# B&R Automation Studio project TD52 (part 112)

#### MsgGTInit.st - Cyclic code
```iecst
(*******************************************************************************
Msg_VE	 			 alarms generation MM_ventilation

This code is confidential and proprietary to the INNIO Company.
It may not be used in any form, or reproduced in any manner,
without written permission of the INNIO Company.
Copyright, INNIO Company, 2019

Customized modifications: -
------------------------

History:
-------
V0.00.0	29.07.2011	lettenb.	new

Instructions for use:
--------------------
1) declare alarm with function block "Msg"

2) use template to create a new alarm, substitue 0000 by message number:

	xMsg0000.Num		:=	0000;					alarm number
	xMsg0000.AmmSysAdr	:=  iAdrAmmBase2MM;			do not change
	xMsg0000.AmmOutAdr	:=  iAdrMM2AmmBase;			do not change

3) 	set alarm number

Outstandings:
------------
(*******************************************************************************)
PROGRAM _INIT

	iAdrAmmBase2MM		:=  ADR(IN_GT.tAB2GT);
	iAdrMM2AmmBase		:=  ADR(OUT_GT.tGT2AB);

	(*---------------------------------------------------------------------------*)
	xMsg1027.Num		:=  1027;
	xMsg1027.AmmInAdr	:=  iAdrAmmBase2MM;
	xMsg1027.AmmOutAdr	:=  iAdrMM2AmmBase;

	xMsg1028.Num		:=  1028;
	xMsg1028.AmmInAdr	:=  iAdrAmmBase2MM;
	xMsg1028.AmmOutAdr	:=  iAdrMM2AmmBase;

	xMsg1029.Num		:=  1029;
	xMsg1029.AmmInAdr	:=  iAdrAmmBase2MM;
	xMsg1029.AmmOutAdr	:=  iAdrMM2AmmBase;

	xMsg1030.Num		:=  1030;
	xMsg1030.AmmInAdr	:=  iAdrAmmBase2MM;
	xMsg1030.AmmOutAdr	:=  iAdrMM2AmmBase;

	xMsg1057.Num		:=  1057;
	xMsg1057.AmmInAdr	:=  iAdrAmmBase2MM;
	xMsg1057.AmmOutAdr	:=  iAdrMM2AmmBase;

	xMsg1058.Num		:=  1058;
	xMsg1058.AmmInAdr	:=  iAdrAmmBase2MM;
	xMsg1058.AmmOutAdr	:=  iAdrMM2AmmBase;

	xMsg1084.Num		:=  1084;
	xMsg1084.AmmInAdr	:=  iAdrAmmBase2MM;
	xMsg1084.AmmOutAdr	:=  iAdrMM2AmmBase;

	xMsg1085.Num		:=  1085;
	xMsg1085.AmmInAdr	:=  iAdrAmmBase2MM;
	xMsg1085.AmmOutAdr	:=  iAdrMM2AmmBase;

	xMsg1086.Num		:=  1086;
	xMsg1086.AmmInAdr	:=  iAdrAmmBase2MM;
	xMsg1086.AmmOutAdr	:=  iAdrMM2AmmBase;

	xMsg1087.Num		:=  1087;
	xMsg1087.AmmInAdr	:=  iAdrAmmBase2MM;
	xMsg1087.AmmOutAdr	:=  iAdrMM2AmmBase;

	xMsg1088.Num		:=  1088;
	xMsg1088.AmmInAdr	:=  iAdrAmmBase2MM;
	xMsg1088.AmmOutAdr	:=  iAdrMM2AmmBase;

	xMsg1094.Num		:=  1094;
	xMsg1094.AmmInAdr	:=  iAdrAmmBase2MM;
	xMsg1094.AmmOutAdr	:=  iAdrMM2AmmBase;

	xMsg1095.Num		:=  1095;
	xMsg1095.AmmInAdr	:=  iAdrAmmBase2MM;
	xMsg1095.AmmOutAdr	:=  iAdrMM2AmmBase;

	xMsg1128.Num		:=  1128;
	xMsg1128.AmmInAdr	:=  iAdrAmmBase2MM;
	xMsg1128.AmmOutAdr	:=  iAdrMM2AmmBase;

	xMsg1251.Num		:=  1251;
	xMsg1251.AmmInAdr	:=  iAdrAmmBase2MM;
	xMsg1251.AmmOutAdr	:=  iAdrMM2AmmBase;

	xMsg1252.Num		:=  1252;
	xMsg1252.AmmInAdr	:=  iAdrAmmBase2MM;
	xMsg1252.AmmOutAdr	:=  iAdrMM2AmmBase;

	xMsg2243.Num		:=  2243;
	xMsg2243.AmmInAdr	:=  iAdrAmmBase2MM;
	xMsg2243.AmmOutAdr	:=  iAdrMM2AmmBase;

	xMsg2246.Num		:=  2246;
	xMsg2246.AmmInAdr	:=  iAdrAmmBase2MM;
	xMsg2246.AmmOutAdr	:=  iAdrMM2AmmBase;

	xMsg2247.Num		:=  2247;
	xMsg2247.AmmInAdr	:=  iAdrAmmBase2MM;
	xMsg2247.AmmOutAdr	:=  iAdrMM2AmmBase;

	xMsg2250.Num		:=  2250;
	xMsg2250.AmmInAdr	:=  iAdrAmmBase2MM;
	xMsg2250.AmmOutAdr	:=  iAdrMM2AmmBase;

	xMsg2251.Num		:=  2251;
	xMsg2251.AmmInAdr	:=  iAdrAmmBase2MM;
	xMsg2251.AmmOutAdr	:=  iAdrMM2AmmBase;

	xMsg2257.Num		:=  2257;
	xMsg2257.AmmInAdr	:=  iAdrAmmBase2MM;
	xMsg2257.AmmOutAdr	:=  iAdrMM2AmmBase;

	xMsg2535.Num		:=  2535;
	xMsg2535.AmmInAdr	:=  iAdrAmmBase2MM;
	xMsg2535.AmmOutAdr	:=  iAdrMM2AmmBase;

	xMsg2536.Num		:=  2536;
	xMsg2536.AmmInAdr	:=  iAdrAmmBase2MM;
	xMsg2536.AmmOutAdr	:=  iAdrMM2AmmBase;

	xMsg2537.Num		:=  2537;
	xMsg2537.AmmInAdr	:=  iAdrAmmBase2MM;
	xMsg2537.AmmOutAdr	:=  iAdrMM2AmmBase;

	xMsg2538.Num		:=  2538;
	xMsg2538.AmmInAdr	:=  iAdrAmmBase2MM;
	xMsg2538.AmmOutAdr	:=  iAdrMM2AmmBase;

	xMsg2578.Num		:=  2578;
	xMsg2578.AmmInAdr	:=  iAdrAmmBase2MM;
	xMsg2578.AmmOutAdr	:=  iAdrMM2AmmBase;

	xMsg2674.Num		:=  2674;
	xMsg2674.AmmInAdr	:=  iAdrAmmBase2MM;
	xMsg2674.AmmOutAdr	:=  iAdrMM2AmmBase;

	xMsg3004.Num		:=  3004;
	xMsg3004.AmmInAdr	:=  iAdrAmmBase2MM;
	xMsg3004.AmmOutAdr	:=  iAdrMM2AmmBase;

	xMsg3153.Num		:=  3153;
	xMsg3153.AmmInAdr	:=  iAdrAmmBase2MM;
	xMsg3153.AmmOutAdr	:=  iAdrMM2AmmBase;

	xMsg3154.Num		:=  3154;
	xMsg3154.AmmInAdr	:=  iAdrAmmBase2MM;
	xMsg3154.AmmOutAdr	:=  iAdrMM2AmmBase;

	xMsg3155.Num		:=  3155;
	xMsg3155.AmmInAdr	:=  iAdrAmmBase2MM;
	xMsg3155.AmmOutAdr	:=  iAdrMM2AmmBase;

	xMsg3156.Num		:=  3156;
	xMsg3156.AmmInAdr	:=  iAdrAmmBase2MM;
	xMsg3156.AmmOutAdr	:=  iAdrMM2AmmBase;

	xMsg3157.Num		:=  3157;
	xMsg3157.AmmInAdr	:=  iAdrAmmBase2MM;
	xMsg3157.AmmOutAdr	:=  iAdrMM2AmmBase;

	xMsg3158.Num		:=  3158;
	xMsg3158.AmmInAdr	:=  iAdrAmmBase2MM;
	xMsg3158.AmmOutAdr	:=  iAdrMM2AmmBase;

	xMsg3159.Num		:=  3159;
	xMsg3159.AmmInAdr	:=  iAdrAmmBase2MM;
	xMsg3159.AmmOutAdr	:=  iAdrMM2AmmBase;

	xMsg3160.Num		:=  3160;
	xMsg3160.AmmInAdr	:=  iAdrAmmBase2MM;
	xMsg3160.AmmOutAdr	:=  iAdrMM2AmmBase;

	xMsg3221.Num		:=  3221;
	xMsg3221.AmmInAdr	:=  iAdrAmmBase2MM;
	xMsg3221.AmmOutAdr	:=  iAdrMM2AmmBase;

	xMsg3222.Num		:=  3222;
	xMsg3222.AmmInAdr	:=  iAdrAmmBase2MM;
	xMsg3222.AmmOutAdr	:=  iAdrMM2AmmBase;

	xMsg3227.Num		:=	3227;
	xMsg3227.AmmInAdr	:=  iAdrAmmBase2MM;
	xMsg3227.AmmOutAdr	:=  iAdrMM2AmmBase;

	xMsg3257.Num		:=	3257;
	xMsg3257.AmmInAdr	:=  iAdrAmmBase2MM;
	xMsg3257.AmmOutAdr	:=  iAdrMM2AmmBase;

	xMsg3258.Num		:=	3258;
	xMsg3258.AmmInAdr	:=  iAdrAmmBase2MM;
	xMsg3258.AmmOutAdr	:=  iAdrMM2AmmBase;

	xMsg3259.Num		:=	3259;
	xMsg3259.AmmInAdr	:=  iAdrAmmBase2MM;
	xMsg3259.AmmOutAdr	:=  iAdrMM2AmmBase;

	xMsg3260.Num		:=	3260;
	xMsg3260.AmmInAdr	:=  iAdrAmmBase2MM;
	xMsg3260.AmmOutAdr	:=  iAdrMM2AmmBase;

	xMsg3261.Num		:=	3261;
	xMsg3261.AmmInAdr	:=  iAdrAmmBase2MM;
	xMsg3261.AmmOutAdr	:=  iAdrMM2AmmBase;

	xMsg3262.Num		:=	3262;
	xMsg3262.AmmInAdr	:=  iAdrAmmBase2MM;
	xMsg3262.AmmOutAdr	:=  iAdrMM2AmmBase;

	xMsg3308.Num		:=  3308;
	xMsg3308.AmmInAdr	:=  iAdrAmmBase2MM;
	xMsg3308.AmmOutAdr	:=  iAdrMM2AmmBase;

	xMsg3309.Num		:=  3309;
	xMsg3309.AmmInAdr	:=  iAdrAmmBase2MM;
	xMsg3309.AmmOutAdr	:=  iAdrMM2AmmBase;

	xMsg3315.Num		:=  3315;
	xMsg3315.AmmInAdr	:=  iAdrAmmBase2MM;
	xMsg3315.AmmOutAdr	:=  iAdrMM2AmmBase;

	xMsg3316.Num		:=  3316;
	xMsg3316.AmmInAdr	:=  iAdrAmmBase2MM;
	xMsg3316.AmmOutAdr	:=  iAdrMM2AmmBase;

	xMsg3317.Num		:=  3317;
	xMsg3317.AmmInAdr	:=  iAdrAmmBase2MM;
	xMsg3317.AmmOutAdr	:=  iAdrMM2AmmBase;

	xMsg3318.Num		:=  3318;
	xMsg3318.AmmInAdr	:=  iAdrAmmBase2MM;
	xMsg3318.AmmOutAdr	:=  iAdrMM2AmmBase;

	xMsg3320.Num		:=  3320;
	xMsg3320.AmmInAdr	:=  iAdrAmmBase2MM;
	xMsg3320.AmmOutAdr	:=  iAdrMM2AmmBase;

	xMsg3324.Num		:=  3324;
	xMsg3324.AmmInAdr	:=  iAdrAmmBase2MM;
	xMsg3324.AmmOutAdr	:=  iAdrMM2AmmBase;

	xMsg3325.Num		:=  3325;
	xMsg3325.AmmInAdr	:=  iAdrAmmBase2MM;
	xMsg3325.AmmOutAdr	:=  iAdrMM2AmmBase;

	xMsg3326.Num		:=  3326;
	xMsg3326.AmmInAdr	:=  iAdrAmmBase2MM;
	xMsg3326.AmmOutAdr	:=  iAdrMM2AmmBase;

	xMsg3327.Num		:=  3327;
	xMsg3327.AmmInAdr	:=  iAdrAmmBase2MM;
	xMsg3327.AmmOutAdr	:=  iAdrMM2AmmBase;

	xMsg3328.Num		:=  3328;
	xMsg3328.AmmInAdr	:=  iAdrAmmBase2MM;
	xMsg3328.AmmOutAdr	:=  iAdrMM2AmmBase;

	xMsg3353.Num		:=  3353;
	xMsg3353.AmmInAdr	:=  iAdrAmmBase2MM;
	xMsg3353.AmmOutAdr	:=  iAdrMM2AmmBase;

	xMsg3354.Num		:=  3354;
	xMsg3354.AmmInAdr	:=  iAdrAmmBase2MM;
	xMsg3354.AmmOutAdr	:=  iAdrMM2AmmBase;

	xMsg3355.Num		:=  3355;
	xMsg3355.AmmInAdr	:=  iAdrAmmBase2MM;
	xMsg3355.AmmOutAdr	:=  iAdrMM2AmmBase;

	xMsg3356.Num		:=  3356;
	xMsg3356.AmmInAdr	:=  iAdrAmmBase2MM;
	xMsg3356.AmmOutAdr	:=  iAdrMM2AmmBase;

	xMsg3357.Num		:=  3357;
	xMsg3357.AmmInAdr	:=  iAdrAmmBase2MM;
	xMsg3357.AmmOutAdr	:=  iAdrMM2AmmBase;

	xMsg3358.Num		:=  3358;
	xMsg3358.AmmInAdr	:=  iAdrAmmBase2MM;
	xMsg3358.AmmOutAdr	:=  iAdrMM2AmmBase;

	xMsg3359.Num		:=  3359;
	xMsg3359.AmmInAdr	:=  iAdrAmmBase2MM;
	xMsg3359.AmmOutAdr	:=  iAdrMM2AmmBase;

	xMsg3360.Num		:=  3360;
	xMsg3360.AmmInAdr	:=  iAdrAmmBase2MM;
	xMsg3360.AmmOutAdr	:=  iAdrMM2AmmBase;

	xMsg3361.Num		:=  3361;
	xMsg3361.AmmInAdr	:=  iAdrAmmBase2MM;
	xMsg3361.AmmOutAdr	:=  iAdrMM2AmmBase;

	xMsg3362.Num		:=  3362;
	xMsg3362.AmmInAdr	:=  iAdrAmmBase2MM;
	xMsg3362.AmmOutAdr	:=  iAdrMM2AmmBase;

	xMsg3363.Num		:=  3363;
	xMsg3363.AmmInAdr	:=  iAdrAmmBase2MM;
	xMsg3363.AmmOutAdr	:=  iAdrMM2AmmBase;

	xMsg3364.Num		:=  3364;
	xMsg3364.AmmInAdr	:=  iAdrAmmBase2MM;
	xMsg3364.AmmOutAdr	:=  iAdrMM2AmmBase;

	xMsg3365.Num		:=  3365;
	xMsg3365.AmmInAdr	:=  iAdrAmmBase2MM;
	xMsg3365.AmmOutAdr	:=  iAdrMM2AmmBase;

	xMsg3520.Num		:=  3520;
	xMsg3520.AmmInAdr	:=  iAdrAmmBase2MM;
	xMsg3520.AmmOutAdr	:=  iAdrMM2AmmBase;

	xMsg3567.Num		:=  3567;
	xMsg3567.AmmInAdr	:=  iAdrAmmBase2MM;
	xMsg3567.AmmOutAdr	:=  iAdrMM2AmmBase;

	xMsg3568.Num		:=  3568;
	xMsg3568.AmmInAdr	:=  iAdrAmmBase2MM;
	xMsg3568.AmmOutAdr	:=  iAdrMM2AmmBase;

	xMsg3569.Num		:=  3569;
	xMsg3569.AmmInAdr	:=  iAdrAmmBase2MM;
	xMsg3569.AmmOutAdr	:=  iAdrMM2AmmBase;

	xMsg3570.Num		:=  3570;
	xMsg3570.AmmInAdr	:=  iAdrAmmBase2MM;
	xMsg3570.AmmOutAdr	:=  iAdrMM2AmmBase;

	xMsg3525.Num		:=  3525;
	xMsg3525.AmmInAdr	:=  iAdrAmmBase2MM;
	xMsg3525.AmmOutAdr	:=  iAdrMM2AmmBase;

	xMsg2247.Num		:=  2247;
	xMsg2247.AmmInAdr	:=  iAdrAmmBase2MM;
	xMsg2247.AmmOutAdr	:=  iAdrMM2AmmBase;

	xMsg2257.Num		:=  2257;
	xMsg2257.AmmInAdr	:=  iAdrAmmBase2MM;
	xMsg2257.AmmOutAdr	:=  iAdrMM2AmmBase;

	xMsg3448.Num		:=  3448;
	xMsg3448.AmmInAdr	:=  iAdrAmmBase2MM;
	xMsg3448.AmmOutAdr	:=  iAdrMM2AmmBase;

	xMsg3444.Num		:=  3444;
	xMsg3444.AmmInAdr	:=  iAdrAmmBase2MM;
	xMsg3444.AmmOutAdr	:=  iAdrMM2AmmBase;

	xMsg3376.Num		:=  3376;
	xMsg3376.AmmInAdr	:=  iAdrAmmBase2MM;
	xMsg3376.AmmOutAdr	:=  iAdrMM2AmmBase;

	xMsg3445.Num		:=  3445;
	xMsg3445.AmmInAdr	:=  iAdrAmmBase2MM;
	xMsg3445.AmmOutAdr	:=  iAdrMM2AmmBase;

	xMsg2289.Num		:=  2289;
	xMsg2289.AmmInAdr	:=  iAdrAmmBase2MM;
	xMsg2289.AmmOutAdr	:=  iAdrMM2AmmBase;

	xMsg2271.Num		:=  2271;
	xMsg2271.AmmInAdr	:=  iAdrAmmBase2MM;
	xMsg2271.AmmOutAdr	:=  iAdrMM2AmmBase;

	xMsg2261.Num		:=  2261;
	xMsg2261.AmmInAdr	:=  iAdrAmmBase2MM;
	xMsg2261.AmmOutAdr	:=  iAdrMM2AmmBase;

	xMsg3377.Num		:=  3377;
	xMsg3377.AmmInAdr	:=  iAdrAmmBase2MM;
	xMsg3377.AmmOutAdr	:=  iAdrMM2AmmBase;

	xMsg2272.Num		:=  2272;
	xMsg2272.AmmInAdr	:=  iAdrAmmBase2MM;
	xMsg2272.AmmOutAdr	:=  iAdrMM2AmmBase;

	xMsg2231.Num		:=  2231;
	xMsg2231.AmmInAdr	:=  iAdrAmmBase2MM;
	xMsg2231.AmmOutAdr	:=  iAdrMM2AmmBase;

	xMsg2240.Num		:=  2240;
	xMsg2240.AmmInAdr	:=  iAdrAmmBase2MM;
	xMsg2240.AmmOutAdr	:=  iAdrMM2AmmBase;

	xMsg2241.Num		:=  2241;
	xMsg2241.AmmInAdr	:=  iAdrAmmBase2MM;
	xMsg2241.AmmOutAdr	:=  iAdrMM2AmmBase;

	xMsg2248.Num		:=  2248;
	xMsg2248.AmmInAdr	:=  iAdrAmmBase2MM;
	xMsg2248.AmmOutAdr	:=  iAdrMM2AmmBase;

	xMsg2249.Num		:=  2249;
	xMsg2249.AmmInAdr	:=  iAdrAmmBase2MM;
	xMsg2249.AmmOutAdr	:=  iAdrMM2AmmBase;

	xMsg2273.Num		:=  2273;
	xMsg2273.AmmInAdr	:=  iAdrAmmBase2MM;
	xMsg2273.AmmOutAdr	:=  iAdrMM2AmmBase;

	xMsg2567.Num		:=  2567;
	xMsg2567.AmmInAdr	:=  iAdrAmmBase2MM;
	xMsg2567.AmmOutAdr	:=  iAdrMM2AmmBase;

	xMsg2568.Num		:=  2568;
	xMsg2568.AmmInAdr	:=  iAdrAmmBase2MM;
	xMsg2568.AmmOutAdr	:=  iAdrMM2AmmBase;

	xMsg2569.Num		:=  2569;
	xMsg2569.AmmInAdr	:=  iAdrAmmBase2MM;
	xMsg2569.AmmOutAdr	:=  iAdrMM2AmmBase;

	xMsg2580.Num		:=  2580;
	xMsg2580.AmmInAdr	:=  iAdrAmmBase2MM;
	xMsg2580.AmmOutAdr	:=  iAdrMM2AmmBase;

	xMsg2581.Num		:=  2581;
	xMsg2581.AmmInAdr	:=  iAdrAmmBase2MM;
	xMsg2581.AmmOutAdr	:=  iAdrMM2AmmBase;

	xMsg2244.Num		:=  2244;
	xMsg2244.AmmInAdr	:=  iAdrAmmBase2MM;
	xMsg2244.AmmOutAdr	:=  iAdrMM2AmmBase;

	xMsg2245.Num		:=  2245;
	xMsg2245.AmmInAdr	:=  iAdrAmmBase2MM;
	xMsg2245.AmmOutAdr	:=  iAdrMM2AmmBase;

	xMsg1265.Num		:=  1265;
	xMsg1265.AmmInAdr	:=  iAdrAmmBase2MM;
	xMsg1265.AmmOutAdr	:=  iAdrMM2AmmBase;

	xMsg1266.Num		:=  1266;
	xMsg1266.AmmInAdr	:=  iAdrAmmBase2MM;
	xMsg1266.AmmOutAdr	:=  iAdrMM2AmmBase;

	xMsg1267.Num		:=  1267;
	xMsg1267.AmmInAdr	:=  iAdrAmmBase2MM;
	xMsg1267.AmmOutAdr	:=  iAdrMM2AmmBase;

	xMsg1268.Num		:=  1268;
	xMsg1268.AmmInAdr	:=  iAdrAmmBase2MM;
	xMsg1268.AmmOutAdr	:=  iAdrMM2AmmBase;

	xMsg1269.Num		:=  1269;
	xMsg1269.AmmInAdr	:=  iAdrAmmBase2MM;
	xMsg1269.AmmOutAdr	:=  iAdrMM2AmmBase;

	xMsg1270.Num		:=  1270;
	xMsg1270.AmmInAdr	:=  iAdrAmmBase2MM;
	xMsg1270.AmmOutAdr	:=  iAdrMM2AmmBase;

	xMsg1271.Num		:=  1271;
	xMsg1271.AmmInAdr	:=  iAdrAmmBase2MM;
	xMsg1271.AmmOutAdr	:=  iAdrMM2AmmBase;

	xMsg1272.Num		:=  1272;
	xMsg1272.AmmInAdr	:=  iAdrAmmBase2MM;
	xMsg1272.AmmOutAdr	:=  iAdrMM2AmmBase;

	xMsg3387.Num		:=  3387;
	xMsg3387.AmmInAdr	:=  iAdrAmmBase2MM;
	xMsg3387.AmmOutAdr	:=  iAdrMM2AmmBase;

	xMsg3388.Num		:=  3388;
	xMsg3388.AmmInAdr	:=  iAdrAmmBase2MM;
	xMsg3388.AmmOutAdr	:=  iAdrMM2AmmBase;

	xMsg3389.Num		:=  3389;
	xMsg3389.AmmInAdr	:=  iAdrAmmBase2MM;
	xMsg3389.AmmOutAdr	:=  iAdrMM2AmmBase;

	xMsg3390.Num		:=  3390;
	xMsg3390.AmmInAdr	:=  iAdrAmmBase2MM;
	xMsg3390.AmmOutAdr	:=  iAdrMM2AmmBase;

	xMsg3391.Num		:=  3391;
	xMsg3391.AmmInAdr	:=  iAdrAmmBase2MM;
	xMsg3391.AmmOutAdr	:=  iAdrMM2AmmBase;

	xMsg3392.Num		:=  3392;
	xMsg3392.AmmInAdr	:=  iAdrAmmBase2MM;
	xMsg3392.AmmOutAdr	:=  iAdrMM2AmmBase;

	xMsg2694.Num		:=  2694;
	xMsg2694.AmmInAdr	:=  iAdrAmmBase2MM;
	xMsg2694.AmmOutAdr	:=  iAdrMM2AmmBase;

	xMsg2695.Num		:=  2695;
	xMsg2695.AmmInAdr	:=  iAdrAmmBase2MM;
	xMsg2695.AmmOutAdr	:=  iAdrMM2AmmBase;

	xMsg2696.Num		:=  2696;
	xMsg2696.AmmInAdr	:=  iAdrAmmBase2MM;
	xMsg2696.AmmOutAdr	:=  iAdrMM2AmmBase;

	xMsg3398.Num		:=  3398;
	xMsg3398.AmmInAdr	:=  iAdrAmmBase2MM;
	xMsg3398.AmmOutAdr	:=  iAdrMM2AmmBase;

	xMsg2753.Num		:=  2753;
	xMsg2753.AmmInAdr	:=  iAdrAmmBase2MM;
	xMsg2753.AmmOutAdr	:=  iAdrMM2AmmBase;

	xMsg2301.Num		:=  2301;
	xMsg2301.AmmInAdr	:=  iAdrAmmBase2MM;
	xMsg2301.AmmOutAdr	:=  iAdrMM2AmmBase;

	xMsg2443.Num		:=  2443;
	xMsg2443.AmmInAdr	:=  iAdrAmmBase2MM;
	xMsg2443.AmmOutAdr	:=  iAdrMM2AmmBase;

	xMsg2444.Num		:=  2444;
	xMsg2444.AmmInAdr	:=  iAdrAmmBase2MM;
	xMsg2444.AmmOutAdr	:=  iAdrMM2AmmBase;

	xMsg2445.Num		:=  2445;
	xMsg2445.AmmInAdr	:=  iAdrAmmBase2MM;
	xMsg2445.AmmOutAdr	:=  iAdrMM2AmmBase;

	xMsg2309.Num		:=  2309;
	xMsg2309.AmmInAdr	:=  iAdrAmmBase2MM;
	xMsg2309.AmmOutAdr	:=  iAdrMM2AmmBase;

	xMsg2462.Num		:=  2462;
	xMsg2462.AmmInAdr	:=  iAdrAmmBase2MM;
	xMsg2462.AmmOutAdr	:=  iAdrMM2AmmBase;

	xMsg2927.Num		:=  2927;
	xMsg2927.AmmInAdr	:=  iAdrAmmBase2MM;
	xMsg2927.AmmOutAdr	:=  iAdrMM2AmmBase;

	xMsg2463.Num		:=  2463;
	xMsg2463.AmmInAdr	:=  iAdrAmmBase2MM;
	xMsg2463.AmmOutAdr	:=  iAdrMM2AmmBase;

	xMsg2465.Num		:=  2465;
	xMsg2465.AmmInAdr	:=  iAdrAmmBase2MM;
	xMsg2465.AmmOutAdr	:=  iAdrMM2AmmBase;

	xMsg2928.Num		:=  2928;
	xMsg2928.AmmInAdr	:=  iAdrAmmBase2MM;
	xMsg2928.AmmOutAdr	:=  iAdrMM2AmmBase;

	xMsg2466.Num		:=  2466;
	xMsg2466.AmmInAdr	:=  iAdrAmmBase2MM;
	xMsg2466.AmmOutAdr	:=  iAdrMM2AmmBase;

	xMsg2467.Num		:=  2467;
	xMsg2467.AmmInAdr	:=  iAdrAmmBase2MM;
	xMsg2467.AmmOutAdr	:=  iAdrMM2AmmBase;

	xMsg2314.Num		:=  2314;
	xMsg2314.AmmInAdr	:=  iAdrAmmBase2MM;
	xMsg2314.AmmOutAdr	:=  iAdrMM2AmmBase;

	xMsg2570.Num		:=  2570;
	xMsg2570.AmmInAdr	:=  iAdrAmmBase2MM;
	xMsg2570.AmmOutAdr	:=  iAdrMM2AmmBase;

	(*BETA V4.07*)
	xMsg2990.Num		:=  2990;
	xMsg2990.AmmInAdr	:=  iAdrAmmBase2MM;
	xMsg2990.AmmOutAdr	:=  iAdrMM2AmmBase;

	xMsg2991.Num		:=  2991;
	xMsg2991.AmmInAdr	:=  iAdrAmmBase2MM;
	xMsg2991.AmmOutAdr	:=  iAdrMM2AmmBase;

	xMsg2992.Num		:=  2992;
	xMsg2992.AmmInAdr	:=  iAdrAmmBase2MM;
	xMsg2992.AmmOutAdr	:=  iAdrMM2AmmBase;

	xMsg2993.Num		:=  2993;
	xMsg2993.AmmInAdr	:=  iAdrAmmBase2MM;
	xMsg2993.AmmOutAdr	:=  iAdrMM2AmmBase;

	xMsg2994.Num		:=  2994;
	xMsg2994.AmmInAdr	:=  iAdrAmmBase2MM;
	xMsg2994.AmmOutAdr	:=  iAdrMM2AmmBase;

	xMsg2995.Num		:=  2995;
	xMsg2995.AmmInAdr	:=  iAdrAmmBase2MM;
	xMsg2995.AmmOutAdr	:=  iAdrMM2AmmBase;

	xMsg2996.Num		:=  2996;
	xMsg2996.AmmInAdr	:=  iAdrAmmBase2MM;
	xMsg2996.AmmOutAdr	:=  iAdrMM2AmmBase;

	xMsg2997.Num		:=  2997;
	xMsg2997.AmmInAdr	:=  iAdrAmmBase2MM;
	xMsg2997.AmmOutAdr	:=  iAdrMM2AmmBase;

	(*BETA V4.07*)
	xMsg9259.Num		:=  9259;
	xMsg9259.AmmInAdr	:=  iAdrAmmBase2MM;
	xMsg9259.AmmOutAdr	:=  iAdrMM2AmmBase;

	xMsg9260.Num		:=  9260;
	xMsg9260.AmmInAdr	:=  iAdrAmmBase2MM;
	xMsg9260.AmmOutAdr	:=  iAdrMM2AmmBase;

	xMsg9275.Num		:=  9275;
	xMsg9275.AmmInAdr	:=  iAdrAmmBase2MM;
	xMsg9275.AmmOutAdr	:=  iAdrMM2AmmBase;

	xMsg9276.Num		:=  9276;					(*Gas Temp max*)
	xMsg9276.AmmInAdr	:=  iAdrAmmBase2MM;
	xMsg9276.AmmOutAdr	:=  iAdrMM2AmmBase;

	xMsg9300.Num		:=  9300;
	xMsg9300.AmmInAdr	:=  iAdrAmmBase2MM;
	xMsg9300.AmmOutAdr	:=  iAdrMM2AmmBase;

	xMsg9301.Num		:=  9301;
	xMsg9301.AmmInAdr	:=  iAdrAmmBase2MM;
	xMsg9301.AmmOutAdr	:=  iAdrMM2AmmBase;

	xMsg9302.Num		:=  9302;
	xMsg9302.AmmInAdr	:=  iAdrAmmBase2MM;
	xMsg9302.AmmOutAdr	:=  iAdrMM2AmmBase;

	xMsg2346.Num		:=  2346;
	xMsg2346.AmmInAdr	:=  iAdrAmmBase2MM;
	xMsg2346.AmmOutAdr	:=  iAdrMM2AmmBase;

	xMsg2976.Num		:=  2976;
	xMsg2976.AmmInAdr	:=  iAdrAmmBase2MM;
	xMsg2976.AmmOutAdr	:=  iAdrMM2AmmBase;

	xMsg9360.Num		:=  9360;
	xMsg9360.AmmInAdr	:=  iAdrAmmBase2MM;
	xMsg9360.AmmOutAdr	:=  iAdrMM2AmmBase;

	xMsg9361.Num		:=  9361;
	xMsg9361.AmmInAdr	:=  iAdrAmmBase2MM;
	xMsg9361.AmmOutAdr	:=  iAdrMM2AmmBase;

	xMsg2364.Num		:=  2364;
	xMsg2364.AmmInAdr	:=  iAdrAmmBase2MM;
	xMsg2364.AmmOutAdr	:=  iAdrMM2AmmBase;

	xMsg9371.Num		:=  9371;
	xMsg9371.AmmInAdr	:=  iAdrAmmBase2MM;
	xMsg9371.AmmOutAdr	:=  iAdrMM2AmmBase;

	xMsg9387.Num		:=  9387;
	xMsg9387.AmmInAdr	:=  iAdrAmmBase2MM;
	xMsg9387.AmmOutAdr	:=  iAdrMM2AmmBase;

	xMsg9086.Num		:=  9086;
	xMsg9086.AmmInAdr	:=  iAdrAmmBase2MM;
	xMsg9086.AmmOutAdr	:=  iAdrMM2AmmBase;

	xMsg9087.Num		:=  9087;
	xMsg9087.AmmInAdr	:=  iAdrAmmBase2MM;
	xMsg9087.AmmOutAdr	:=  iAdrMM2AmmBase;

	xMsg9509.Num		:=  9509;
	xMsg9509.AmmInAdr	:=  iAdrAmmBase2MM;
	xMsg9509.AmmOutAdr	:=  iAdrMM2AmmBase;

	(* template
	xMsg.Num		:=	;
	xMsg.AmmInAdr	:=  iAdrAmmBase2MM;
	xMsg.AmmOutAdr	:=  iAdrMM2AmmBase;
	*)

END_PROGRAM
```

#### MsgGT.var
```iecst
VAR
	iAdrAmmBase2MM : UDINT;
	iAdrMM2AmmBase : UDINT;
	xGRMAX_T_PCGAfCo_Hi : GR_MAXR;
	xGR_MAX_LDR : GR_MAXR;
	xMsg1027 : Msg;
	xMsg1028 : Msg;
	xMsg1029 : Msg;
	xMsg1030 : Msg;
	xMsg1057 : Msg;
	xMsg1058 : Msg;
	xMsg1084 : Msg;
	xMsg1085 : Msg;
	xMsg1086 : Msg;
	xMsg1087 : Msg;
	xMsg1088 : Msg;
	xMsg1094 : Msg;
	xMsg1095 : Msg;
	xMsg1128 : Msg;
	xMsg1251 : Msg;
	xMsg1252 : Msg;
	xMsg1265 : Msg;
	xMsg1266 : Msg;
	xMsg1267 : Msg;
	xMsg1268 : Msg;
	xMsg1269 : Msg;
	xMsg1270 : Msg;
	xMsg1271 : Msg;
	xMsg1272 : Msg;
	xMsg2231 : Msg;
	xMsg2240 : Msg;
	xMsg2241 : Msg;
	xMsg2243 : Msg;
	xMsg2244 : Msg;
	xMsg2245 : Msg;
	xMsg2246 : Msg;
	xMsg2247 : Msg;
	xMsg2248 : Msg;
	xMsg2249 : Msg;
	xMsg2250 : Msg;
	xMsg2251 : Msg;
	xMsg2257 : Msg;
	xMsg2261 : Msg;
	xMsg2271 : Msg;
	xMsg2272 : Msg;
	xMsg2273 : Msg;
	xMsg2289 : Msg;
	xMsg2535 : Msg;
	xMsg2536 : Msg;
	xMsg2537 : Msg;
	xMsg2538 : Msg;
	xMsg2567 : Msg;
	xMsg2568 : Msg;
	xMsg2569 : Msg;
	xMsg2578 : Msg;
	xMsg2580 : Msg;
	xMsg2581 : Msg;
	xMsg2674 : Msg;
	xMsg2694 : Msg;
	xMsg2695 : Msg;
	xMsg2696 : Msg;
	xMsg3004 : Msg;
	xMsg3153 : Msg;
	xMsg3154 : Msg;
	xMsg3155 : Msg;
	xMsg3156 : Msg;
	xMsg3157 : Msg;
	xMsg3158 : Msg;
	xMsg3159 : Msg;
	xMsg3160 : Msg;
	xMsg3221 : Msg;
	xMsg3222 : Msg;
	xMsg3227 : Msg;
	xMsg3257 : Msg;
	xMsg3258 : Msg;
	xMsg3259 : Msg;
	xMsg3260 : Msg;
	xMsg3261 : Msg;
	xMsg3262 : Msg;
	xMsg3308 : Msg;
	xMsg3309 : Msg;
	xMsg3315 : Msg;
	xMsg3316 : Msg;
	xMsg3317 : Msg;
	xMsg3318 : Msg;
	xMsg3320 : Msg;
	xMsg3324 : Msg;
	xMsg3325 : Msg;
	xMsg3326 : Msg;
	xMsg3327 : Msg;
	xMsg3328 : Msg;
	xMsg3353 : Msg;
	xMsg3354 : Msg;
	xMsg3355 : Msg;
	xMsg3356 : Msg;
	xMsg3357 : Msg;
	xMsg3358 : Msg;
	xMsg3359 : Msg;
	xMsg3360 : Msg;
	xMsg3361 : Msg;
	xMsg3362 : Msg;
	xMsg3363 : Msg;
	xMsg3364 : Msg;
	xMsg3365 : Msg;
	xMsg3376 : Msg;
	xMsg3377 : Msg;
	xMsg3387 : Msg;
	xMsg3388 : Msg;
	xMsg3389 : Msg;
	xMsg3390 : Msg;
	xMsg3391 : Msg;
	xMsg3392 : Msg;
	xMsg3444 : Msg;
	xMsg3445 : Msg;
	xMsg3448 : Msg;
	xMsg3520 : Msg;
	xMsg3525 : Msg;
	xMsg3567 : Msg;
	xMsg3568 : Msg;
	xMsg3569 : Msg;
	xMsg3570 : Msg;
	xMsg3398 : Msg;
	xMsg2753 : Msg;
	xMsg2443 : Msg;
	xMsg2444 : Msg;
	xMsg2445 : Msg;
	xMsg2309 : Msg;
	xTOF_UW_VKDR : TOF;
	xTON_UW_PDIFF : TON;
	xMsg2301 : Msg;
	xMsg2462 : Msg;
	xMsg2927 : Msg;
	xTP_2927_from2462 : TP;
	xTP_2927_EngStart : TP;
	xMsg2463 : Msg;
	xMsg2465 : Msg;
	xMsg2928 : Msg;
	xTP_2928_from2465 : TP;
	xTP_2928_EngStart : TP;
	xMsg2466 : Msg;
	xMsg2467 : Msg;
	xMsg2314 : Msg;
	xMsg2570 : Msg;
	tiTON_UW_PDIFF : TIME := 0;
	xMsg9086 : Msg; (*Gas valves open*)
	xMsg9087 : Msg; (*Gas valves closed*)
	xTP_9087_GVOff : TP; (*Gas valves closed*)
	xMsg9259 : Msg;
	xMsg9260 : Msg;
	xMsg9275 : Msg;
	xMsg9276 : Msg;
	xMsg2990 : Msg;
	xMsg2991 : Msg;
	xMsg2992 : Msg;
	xMsg2993 : Msg;
	xMsg2994 : Msg;
	xMsg2995 : Msg;
	xMsg2996 : Msg;
	xMsg2997 : Msg;
	xMsg9300 : Msg;
	xMsg9301 : Msg;
	xMsg9302 : Msg;
	xMsg2346 : Msg;
	xMsg2976 : Msg;
	xMsg9360 : Msg;
	xMsg9361 : Msg;
	xMsg2364 : Msg;
	xMsg9371 : Msg;
	xMsg9387 : Msg;
	xMsg9509 : Msg;
END_VAR
```

### Program Logical/Gastrain/ParGT (IEC) - + Parameter handling

- perm_par.st (not readable text: treated as protected, skipped)

#### perm_par.var
```iecst
VAR
	tParaIntern : ParaHandler_typ; (*Connector type to perm_par*)
	tMM2ParaBase_ReadBack : MM2ParaBase_type; (*INTERNAL! V4.06 new readback structure for information from previous tasks*)
	bWriteDataObj : BOOL; (* TRUE=write data object module *)
	bDataObjLenErr : BOOL; (*Error occured in permem: data module size missmatch*)
	bCreateDataObj : BOOL; (* TRUE=create new data object *)
	bWriteOnce : BOOL; (* write permanent memory once *)
	DatObjCreate_01 : DatObjCreate; (* data object create *)
	DatObjInfoBak_02 : DatObjInfo; (* data object info *)
	DatObjDelete_01 : DatObjDelete; (* data object delete *)
	DatObjRead_01 : DatObjRead; (* data object read *)
	DatObjRead_02 : DatObjRead; (* manual initiated data object read *)
	DatObjWrite_01 : DatObjWrite; (* data object write *)
	DatObjDelete_02 : DatObjDelete; (* data object delete *)
	DatObjDelete_11 : DatObjDelete; (*Delete Backup File*)
	DatObjInfo_01 : DatObjInfo; (* data object info *)
	DatObjInfo_02 : DatObjInfo; (* data object info *)
	szModuleName : STRING[35]; (* module name of object *)
	szModuleNameBackup : STRING[35]; (* module name of posiibly created backup object *)
	DatObjCopy_01 : DatObjCopy;
	bCopyDataObj : BOOL;
	TON_WarnDelay : TON;
	TON_WritePMEM : TON; (* delay write permanent memory *)
	ulPMPointer : UDINT; (* adress of actual checksum value *)
	ulChecksum : UDINT; (* parameter checksum value *)
	pm_len : UDINT; (* permanent value lenght *)
	ulChecksumOld : UDINT; (* last vlaue of parameter checksum *)
	ulChkValue : UDINT; (* actual value of parameter pointer *)
	pm_id : UDINT; (* permanent value identifier *)
	pm_p : UDINT; (* permanent value pointer *)
	DatObjInfo_META : DatObjInfo;
	DatObjRead_META : DatObjRead;
	szMetaDataRaw : STRING[2000];
	szMetaData : ARRAY[0..4] OF STRING[35];
	szMetaDataVis : ARRAY[0..3] OF STRING[35];
	ssIndex : INT;
	ssCount : INT;
	ucMetaDataRaw : ARRAY[0..2000] OF USINT;
	ssCount2 : INT;
	szMetaDataFile : STRING[10];
	szText1 : STRING[20];
	pv_adr_IN_XX_tPB2MM : UDINT;
	pv_lng : UDINT;
	pv_lng_IN_XX_tPB2MM : UDINT;
	pv_lng_OUT_XX_tPB2MM : UDINT;
	szText2 : STRING[20];
	pv_adr_OUT_XX_tXX2PB : UDINT;
END_VAR
VAR CONSTANT
	ERR_NOERROR : UINT := 0;
END_VAR
VAR
	usPMWriteCnt : UINT;
	pm_Error : UDINT; (* permanent value error *) (* Deleted: pm : ParaMem_typ; permanent memory tags mathias, 22.8.11*)
	fun_Error : UDINT := 0; (*state > 0 = function error*)
	xLocalParaCheck : ParaCheckFUB; (*local function instance to check parameter values*)
	TON_ParaSetupOk : TON;
	bParaCheckSystemOk : BOOL;
	iDebug_ParaOkChecked : UDINT;
	bRestoreBackupDataObj : BOOL := FALSE;
	bRestoreDataObjContent : BOOL := FALSE;
	pm_id_backup : UDINT;
	pm_p_Backup : UDINT;
	DatObjCopy_02 : DatObjCopy;
	bDeleteBackupDataObj : BOOL := FALSE; (*Command to delete backup data module file on purpose*)
	bDebugPara : ARRAY[0..5] OF BOOL;
	ssIndex2 : INT;
	ssIndex3 : INT;
	ssIndex4 : INT;
	ssIndexVis : INT;
	szText : STRING[40];
	pv_adr_Para : UDINT;
	szParaSnippet : ARRAY[0..5] OF STRING[150];
	szParaIndex : STRING[10];
	slValue : DINT;
	iModuleDLD_ResetCount : INT;
	bDownloadDetected : BOOL;
	bFlagParaStructCopyWorking : BOOL; (*true, if cyclic para copying is active, 1 false cycle at every copy *)
	bStoreInitParaInDataObj : BOOL := FALSE;
	bTestflag : BOOL;
	bReadOutMETA_Once : BOOL;
	tParaCheck_iPvAdress : ARRAY[0..5] OF UDINT;
	tParaCheck_iPvLengt : ARRAY[0..5] OF UDINT;
	tParaCheck_rPvValue : ARRAY[0..5] OF REAL;
	tParaCheck_rRangeMIN : ARRAY[0..5] OF REAL;
	tParaCheck_rRangeMAX : ARRAY[0..5] OF REAL;
	tParaCheck_szPvName : ARRAY[0..5] OF STRING[35];
	ssFormatDetected : INT;
	szMetaDataPart : STRING[150];
	szFullTaskName : STRING[35];
	szFullMetaModuleName : STRING[35];
	debugLen : INT;
	debugSize : INT := 0;
	strcat_adr1 : UDINT;
	strcat_adr2 : UDINT;
	ssIndexTN : INT;
	bAlternate : BOOL;
	n : INT;
	iAlternateChecksum : DINT;
	iAlternateChecksumOld : DINT;
	ulDebugChkValue : ARRAY[0..999] OF UDINT;
	Adr1 : UDINT;
	Adr2 : UDINT;
	usPMWriteCntStepsize : UINT := 1; (*different step sizes to help debug*)
	usPMWriteCntXOR : UINT;
	usPMWriteCntAltSum : UINT;
	ulAdrPM : UDINT;
	usChkValuePM : USINT;
	ulAdrPara : UDINT;
	ulPara_len : UDINT;
	usChkValuePara : USINT;
	iDebugCountPMDifferences : DINT := 0;
	bEngineRunDetected : BOOL; (*detection status bit autocommand 100 /101  for engine run state*)
	ucMetaDataDebugInfoLine : ARRAY[0..24] OF STRING[80];
	ssIndexMand : INT := 0;
	szMetaDataMand : STRING[35];
	iMyErrorInfo_Autoreset : DINT; (*internal autoreset counter*)
	ssIndex_Version : INT; (*internal*)
	ssIndex_BU : INT; (*internal*)
	ssIndex_BU2 : INT; (*internal*)
END_VAR
```

### Program Logical/Gastrain/PermGT (IEC) - + Permanent stored data

- PermGTInit.st (not readable text: treated as protected, skipped)

- PermGTCyclic.st (not readable text: treated as protected, skipped)

#### PermGT.var - Lokale Variablen
```iecst
VAR
	pm_Error : UINT;
	write_once : BOOL;
	pm_len : UDINT;
	ModulName : STRING[35];
	DatObjInfo_01 : DatObjInfo;
	pm_id : UDINT;
	pm_p : UDINT;
	bCreateDataObj : BOOL;
	perm_par_vers : UINT;
	DatObjRead_01 : DatObjRead;
	DatObjDelete_PermMem : DatObjDelete;
	DatObjCreate_01 : DatObjCreate;
	DatObjWrite_01 : DatObjWrite;
	ulChecksumOld : UDINT;
	ulPMPointer : UDINT;
	ulChkValue : UDINT;
	TON_WritePMEM : TON;
	ulChecksum : UDINT;
	bWriteDataObj : BOOL;
	TON_WarnDelay : TON;
END_VAR
VAR CONSTANT
	ERR_NOERROR : UINT := 0;
END_VAR
VAR
	pmm : PERM_GT_struct;
	TON_BlockMinFileAge : TON; (*waiting time without file write after successful performed write*)
	bBlock_MinFileAge : BOOL := FALSE; (*pause the perm file write after each sucessful write*)
	iPM_WriteCnt : UDINT; (* *) (*old VarName: usPMWriteCnt*)
END_VAR
```

### Program Logical/Gastrain/PermGT2 (IEC) - + Permanent stored data 2

- PermGT2Init.st (not readable text: treated as protected, skipped)

- PermGT2Cyclic.st (not readable text: treated as protected, skipped)

#### PermGT2.var - Lokale Variablen
```iecst
VAR
	pm_Error : UINT;
	write_once : BOOL;
	pm_len : UDINT;
	ModulName : STRING[35];
	DatObjInfo_01 : DatObjInfo;
	pm_id : UDINT;
	pm_p : UDINT;
	bCreateDataObj : BOOL;
	perm_par_vers : UINT;
	DatObjRead_01 : DatObjRead;
	usPMWriteCnt : UINT;
	DatObjDelete_PermMem : DatObjDelete;
	DatObjCreate_01 : DatObjCreate;
	DatObjWrite_01 : DatObjWrite;
	ulChecksumOld : UDINT;
	ulPMPointer : UDINT;
	ulChkValue : UDINT;
	TON_WritePMEM : TON;
	ulChecksum : UDINT;
	bWriteDataObj : BOOL;
	TON_WarnDelay : TON;
END_VAR
VAR CONSTANT
	ERR_NOERROR : UINT := 0;
END_VAR
VAR
	pmm2 : PERM_GT2_struct;
END_VAR
```

### Program Logical/Gastrain/VisGT (IEC) - Visualization task for Gas train module

#### VisGTCyclic.st - Cyclic code
```iecst
(*******************************************************************************
VisGT	 			 VISU variables

This code is confidential and proprietary to the INNIO Company.
It may not be used in any form, or reproduced in any manner,
without written permission of the INNIO Company.
Copyright, INNIO Company, 2025

Customized modifications: -
------------------------

History:
-------
V04.00.00	19.06.2012	Denk	 	new
V04.00.01	21.02.2014	Zengerer	iIdx_SelGasTyp TESTBENCH MODIFICATION because of OPC UA troubles
V04.00.01	12.03.2014	Zengerer	Bugfix version
V04.00.02	13.05.2014	Denk		MM2VIS.rPr_PCGT added
V04.03.00  	13.11.2014  Mari 		Porting J920 for XT4
			11.02.2015	Denk		MM2VIS.rT_PCGT, MM2VIS.rPr_PCGT_a_Filt added
			01.04.2015	Denk		MM2VIS.rT_GR := IN_GT.tT_GR.Ai; added
			02.06.2015  Denk		MM2VIS.rPr_PCGT_sp, MM2VIS.rPr_MGT_sp now in gas_train task
V04.05.00   29.08.2017  Denk		MM2VIS.rT_PCGAfCo added
V04.06.00   20.09.2018  Perktold	MM2VIS.bGT_FS_Release added
V04.07.00	15.02.2019	Denk		Bugfix, when parameter 11363 is TRUE, AutGas was not active after PLC warmstart.
V04.09.00	27.06.2019	Denk		Additional measurements in natural gas train (T_GT_NG, Pr_GT_NG, Vol_GT_NG)
V04.12.00	22.01.2023	Zuschnig	Add filtered H2 content
V04.25.00	30.12.2025	Tinello		Logic modified because of SafetyPLC

Instructions for use:
--------------------

Outstandings:
------------

(*******************************************************************************)

PROGRAM _CYCLIC

	(* Module 2 VISU *)
	MM2VIS.bGasMixingActive 	:= OUT_GT.bGasMixingActive;
	MM2VIS.bGT1_SafeDevice  	:= OUT_GT.tGT1_SafeDevice.Do OR IN_GT.bSafeOUT_GT1_SD_Dem_PS;		(* SAFETY PLC *)
	MM2VIS.bGT2_SafeDevice  	:= OUT_GT.tGT2_SafeDevice.Do OR IN_GT.bSafeOUT_GT2_SD_Dem_PS;		(* SAFETY PLC *)
	MM2VIS.rGT_QualMix_1_2   	:= OUT_GT.rGT_QualMix_1_2;
	MM2VIS.rP_Red_CH4_Norm   	:= OUT_GT.rP_Red_CH4_Norm;
	MM2VIS.rP_Red_CV_Norm    	:= OUT_GT.rP_Red_CV_Norm;
	MM2VIS.rP_Red_GasPr_Norm 	:= OUT_GT.rP_Red_GasPr_Norm;
	MM2VIS.bGT1_FailureTest		:= M_STGAS1;
	MM2VIS.bGT2_FailureTest		:= M_STGAS2;
	MM2VIS.bGV1_Open			:= OUT_GT.tGV1_Open.Do;
	MM2VIS.bGV2_Open			:= OUT_GT.tGV2_Open.Do;
	MM2VIS.bPCG_GV_Open			:= OUT_GT.tPCG_GV_Open.Do;
	MM2VIS.bPCG_BPV_Open		:= OUT_GT.tPCG_BPV_Open.Do;
	MM2VIS.bGT1_CheckOK			:= OUT_GT.bGT1_CheckOK;
	MM2VIS.bGT2_CheckOK			:= OUT_GT.bGT2_CheckOK;
	MM2VIS.bGT_FS_Release		:= OUT_GT.bGT1_SafeDevOK AND OUT_GT.bGT2_SafeDevOK AND OUT_GT.bPCGT_SafeDevOK;
	MM2VIS.rGT_RatioMix			:= OUT_GT.rGT_RatioMix;
	MM2VIS.rP_Red_Pr_PCGT_Norm	:= OUT_GT.rP_Red_Pr_PCGT_Norm;
	MM2VIS.bSelGasTyp1			:= OUT_GT.bSelGasTyp1;
	MM2VIS.bSelGasTyp2			:= OUT_GT.bSelGasTyp2;
	MM2VIS.bSelGasTyp3			:= OUT_GT.bSelGasTyp3;
	MM2VIS.bSelGasTyp4			:= OUT_GT.bSelGasTyp4;
	MM2VIS.bSelGasTyp0			:= OUT_GT.bSelGasTyp0;
	MM2VIS.bSelGasTypAut 		:= OUT_GT.bSelGasTypAut;
	MM2VIS.bSelGasTypMix		:= OUT_GT.bSelGasTypMix;
	IF OUT_GT.iIdx_Gtyp_Dem > 0 THEN
		MM2VIS.iIdx_Gtyp_Dem	:= OUT_GT.iIdx_Gtyp_Dem;
	ELSE
		IF bCrossOver THEN
			MM2VIS.iIdx_Gtyp_Dem := 5;
			IF OUT_GT.bGT_Ipol12Active THEN
				MM2VIS.iIdx_Gtyp_Dem := 6;
			END_IF
		END_IF
	END_IF
	MM2VIS.bGV_On				:= (OUT_GT.bGV_On 			AND NOT IN_GT.bSafetyPLC_Active) OR 	(* SAFETY PLC *)
								   (IN_GT.bSafeOUT_GV_Open	AND		IN_GT.bSafetyPLC_Active);		(* SAFETY PLC *)
	MM2VIS.rPr_PC_Diff			:= ANA_PDIFF;
	MM2VIS.rPr_PCGT				:= IN_GT.tPr_PCGT.Ai;
	MM2VIS.rPr_PCGT_a_Filt		:= IN_GT.tPr_PCGT.Ai;
	MM2VIS.rDPr_PCGT_SetAct		:= rDPr_PCGT_SetAct;
	MM2VIS.rDPr_MGT_SetAct 		:= rDPr_MGT_SetAct;
	MM2VIS.rPr_MGT_Out_Calc		:= rPr_MGT_Out_Calc;
	MM2VIS.rPr_GR_Avg			:= rPr_GR_Avg;
	MM2VIS.rPr_PCGT_Out			:= IN_GT.tPr_PCGT_Out.Ai;
	MM2VIS.rPr_MGT_a_Filt		:= IN_GT.tPr_MGT_a_Filt.Ai;
	MM2VIS.bMGT_BOV				:= OUT_GT.tMGT_BOV.Do;
	MM2VIS.rPr_MGT_Diff			:= rPr_MGT_Diff;
	MM2VIS.rT_PCGAfCo   		:= IN_GT.tT_PCGAfCo.Ai;
	MM2VIS.rGT_H2 				:= xLCRPT1_H2.y;

	(* from HalIO *)
	MM2VIS.rGT_CH4 			:= rGT_CH4;
	MM2VIS.rGT_CV  			:= rGT_CV;
	MM2VIS.rGT_O2 			:= IN_GT.tGT_O2.Ai;
	MM2VIS.rPr_PCG 			:= IN_GT.tPr_PCG.Ai;
	MM2VIS.rT_GT 			:= IN_GT.tT_GT.Ai;
	MM2VIS.rVol_GT 			:= IN_GT.tVol_GT.Ai;
  	MM2VIS.rPr_GT_Gas       := IN_GT.tPr_GT_Gas.Ai;
	MM2VIS.rPr_GT_Suct      := IN_GT.tPr_GT_Suct.Ai;
	MM2VIS.rPr_PC			:= IN_GT.tPr_PC.Ai;
	MM2VIS.rT_PCGT			:= IN_GT.tT_PCGT.Ai;
	MM2VIS.rT_GR 			:= IN_GT.tT_GR.Ai;
	MM2VIS.rT_GT_NG			:= IN_GT.tT_GT_NG.Ai;
	MM2VIS.rPr_GT_NG		:= IN_GT.tPr_GT_NG.Ai;
	MM2VIS.rVol_GT_NG		:= IN_GT.tVol_GT_NG.Ai;

	(* VISU 2 Module *)
	IF EDGEPOS(Para.bGT_AutGas_Ena) THEN	(* Presetting of AutGas when parameter 11363 is TRUE *)
		VIS2MM.iIdx_SelGasTyp := 7;
 	END_IF;
	iIdx_SelGasTyp       	:= VIS2MM.iIdx_SelGasTyp;
	bGT_MixingEna        	:= VIS2MM.bGT_MixingEna;
	bGT_QualMix_Man_Set  	:= VIS2MM.bGT_QualMix_Man_Set;
	bGT_RatioMix_Man_Set 	:= VIS2MM.bGT_RatioMix_Man_Set;
	rGT_QualMix_Man_Set  	:= VIS2MM.rGT_QualMix_Man_Set;
	rGT_RatioMix_Man_Set 	:= VIS2MM.rGT_RatioMix_Man_Set;

END_PROGRAM
```

#### VisGTInit.st - Initialization code
```iecst
(********************************************************************
 * COPYRIGHT -- INNIO Company
 ********************************************************************
 * Program: VisGT
 * File: VisGTInit.st
 * Author: 105051626
 * Created: July 05, 2012
 ********************************************************************
 * Implementation of program VisGT
 ********************************************************************)

PROGRAM _INIT

	(*Predefine gastype 1, if nothing else is selected*)
	IF VIS2MM.iIdx_SelGasTyp = 0 THEN
		VIS2MM.iIdx_SelGasTyp	:= 1;
	END_IF

END_PROGRAM
```

### Package Logical/HalIO - HA: Hardware Abstraction Layer for Inputs/Outputs

### Data object Logical/HalIO/META_HA (Simple) - HalIO META data module

#### META_HA.dat
```
; *******************************************************************************
; AGGR: Module Meta Data (data module)
;
; This code is confidential and proprietary to the INNIO Company.
; It may not be used in any form, or reproduced in any manner, without the express
; written permission of the INNIO Company.
; Copyright, INNIO Company, 2025
;
; Customized modifications: -
; ------------------------
;
; History:
; -------
; V3.99	  06-03-2013	Weitzer, generated for modular software
; 		  06-06-2013	Zengerer structure prototype according to todays meeting
; V4.00   31-01-2014	Weitzer, versions changed
; V4.01   22-07-2014	Weitzer, add new IO channels
; V4.01.1 10-10-2014	Weitzer, correction of IO channel monitoring
; V4.03	  14-01-2015	Weitzer, new IOs added for J920
;								 add engine version information
; V4.03.1 11.06.2015	Zengerer version + dependencies changed (IF change with array index 0 for compatibility with c-tasks)
; V4.03.2 03-03-2016	Weitzer, add engine speed at IN_HA for F = 0Hz at engine stop
; V4.04.0 01.06.2016	Tinello, CM&U Sensor package added
; V4.05.0 01.06.2016	lettenb. faststart IO added;
;		  18.07.2017	Messner, Oil circuit fast start V2
;		  07.08.2017	Messner, Starter battery voltage monitoring
;		  20.09.2017	Messner, Active Cooling Program added
;		  27.07.2017	Messner, CAN Diagnosis Picture added
;		  04.12.2017	Messner, Oxidation catalyst added
; V4.05.1 14.02.2018	Weitzer, EOP_BWS2 added, correct CAN diagnosis data
;         22.02.2018	lettenb. AI_PF_CosPCtr_Set removed, dependancies
; V4.05.2 19.03.2018	Denk, 	 WinMOD simulation ON/OFF logic added
; V4.05.3 26.03.2018	Farre, 	 Signals removed (PF_CosPCtr_PF1_Ena, PF_CosPCtr_PF2_Ena, PF_CosPCtr_PF3_Ena, PF_CosPCtr_PF4_Ena, PF_CosPCtr_PF5_Ena)
; V4.06.0 01.03.2018	Perktold, I/Os for (very)fast start added
;         16.03.2018	502423184 ".Exist" added to HALioBase library for analog inputs
;	  	  11.10.2018	Schmid,	 module identifiers for coated modules included
; V4.07.0 12.07.2018	502423184,	added G2  (see details in section Info below, add new info there!)
; V4.08.0 07.02.2019	Schmid,  B&R IPC PPC3100 adaptations (PLC address for CAN device changed)
; V4.08.1 26.11.2019	Denk,  Exception task for cycle time violation TC#1 added
; V4.08.2 10.12.2019	Schmid,  MMD over- and undervoltage protection: changed monitoring to phase-phase voltages
; V4.09.0 12.12.2019	Tinello, CAN NOx infos added for HMI
;		  17.12.2019	Schmid,	 new scaling parameters, IOs, MMU parameter
; V4.09.1 16.04.2020	Schmid,	 bugfix: spare analog input (CustAnaIn) scaling corrected to allow falling slope
;         25.06.2020	lettenb. X20CM985-1_fw_upgrade(1.9.0.0 -> 2.2.0.0)
; V4.10.0 20.07.2020	Schmid,	 new scaling parameters, IOs
;		  21.10.2020	lettenb. Pr_Oxicat_In/Out Filter 0 -> 1000 (1s), bu
; V4.10.0 03.11.2020	Schmid,  additional CAN node interfaces for engine and NOx sensor CAN
;		  12.11.2020	lettenb. DI: Dem_EU_Block2, tDem_EU_Block3 added
; V4.10.1 27.04.2021	Schmid,  bugfix: corrected Cnt_N_AirStarter memory interference issue (AI_INT32 to AI_INT16)
; 		  10.05.2021	Weitzer	 System cyclic time viaolation monitoring added
; V4.10.2 12.05.2021	Schmid	 bugfix: corrected scaling and GoodQual limits for U_SetExt_Norm
; V4.11.0 17.08.2021	Weitzer	 UR20 IO system added
;		  29.11.2021	lettenb. IOs for GR added
; 		  07.12.2021	Schmid	 flexible CAN interface detection
;		  22.12.2021	Andre,	 caninitHA: avoid potential array index overrun
; V4.12.0 29.06.2022	lettenb. IOs added
;		  06.09.2022	Keller	 change mapping OUT_OP.tLSL_out to TC2
;		  28-10-2022	Weitzer, added auto detect multiplier for bus bar and synch voltages > 30kV
;		  13-12-2022	Schmidt, switch to separate sync window settings if fast-sync active
;		  02.12.2022	Weitzer, add IGN2 CAN interface
; 		  22.01.2023	Zuschnig H2 content added
; V4.13.0 26.05.2023	Zuschnig Added standardized AI input for gas mixing ratio
;		  27.09.2023 	Bacci	 Flucon sensor clean-up
;		  17.10.2023	Andre	 Only perform ARwin warm start if the CAN bus off state cannot be quit
;		  21.11.2023	Tinello	 Added urea tank level
;         21.11.2023    Heim Markus add hardware parameters for ctr 9,10,11,12,14,15,16,17,21,22,23,24,25,26,27,30,31,34
;		  28.11.2023	Maran	 added IOs for thermal reactor auxiliary gas injection monitoring
;		  30.11.2023	Farre, 	 added ILF (de)activation bits
;		  22.01.2024	Astner	 OpcUA Pub/Sub Plant Communication added (Dependency SY 4.13)
;         23.02.2024    Astner   Added Configuration of ModbusTCP ethernet interfaces on X20 CPU
;		  05.03.2024	Bacci	 Added hardware bypass digital twin - T3 adaptive cranking time
;		  07.03.2024	Farre	 issue #890, #1089: re-define settings and scale analog input signals sent to GR and GC
; V4.14.0 28.03.2024	Soto/Farre,	CAN NOx IF1 shared with Wastegate, interfaces duplicated (2023-174)
; 		  18.06.2024	Soto	 added CAN interface for Low NOx sensor IF3 (2023-183)
; 		  07.10.2024	Kafka	 Remove G2 signals, SAFI / KLS21 devices of bank B use 2nd CAN card and the rest use 1st one
;		  08.11.2024	Bacci	 Added cold country antifreeze arrangements (2020-25)
;		  18.11.2024	Farre	 send to MMU1 current asymmetry value from a new parameter (2024-234)
;		  19.11.2024	Farre	 added auto detect multiplier for grid voltage (2024-236)
;		  21.11.2024	Farre	 additional moisture sensor in air line CEMS (2023-183)
;		  22.11.2024	Schmidt	 Added IO for pre chamber gas bypass valve
;		  25.11.2024	Zengerer Multi analog temp input variants issue #1706 - T_HW_Re, T_HW_ReAfEC, T_HW_Su ...
;		  28.11.2024	Astner	ANSL Plant Communication added (Dependency MSY 4.09)
;		  29.11.2024	Zengerer new EO_FreshOilPump & EO_WasteOilPump DO
; 		  26.02.2025	Tinello	 Added SafetyPLC
;		  07.02.2025	add possibility for customized mains settings for MMD1 and MMD2
; V4.25.0 26.11.2025	Bacci	 Safety Function - Insufficient Ventilation (2024-202): ERV digital feedback added
; 		  10.07.2025	Tinello	 SafetyPLC Phase II added
;
; Instructions for use:
; --------------------
; make only changes at the version numbers
; watch out for proper "" and <> </> marks and use := and = on the right places!
;
; Outstandings:
; ------------
; datamodule syntax checker
; (caution: syntax errors here may cause plc runtime errors!)
;
; *******************************************************************************
;
"<META>"
;
; Module ID
"<MODUL>HA</MODUL>"
;
; Module Version (xx.yy.zz.cc)
"<VERSION>04.25.00.00</VERSION>"
;
; Module Basisupdate Version BU (00-99)
"<BASISUPDATE_VERSION>00</BASISUPDATE_VERSION>"
;
; Specify order number
"<ORDER>DT52</ORDER>"  				;<!--PLEASE FILL IN ORDER ID (HAL_IO is allways customized)-->
;
; Specify engine type
"<ENGINE_TYPE>624</ENGINE_TYPE>"	;<!--PLEASE FILL IN ENGINE TYPE-->
;
; Specify engine version
"<ENGINE_VERSION>L3785</ENGINE_VERSION>" ;<!--PLEASE FILL IN ENGINE VERSION-->
;
; Parameter Check <PARAn Name='aAbcdef' MIN='xxx' MAX='yyy' />  (watch for correct spacings and apostrophs!)
"<PARAMETER_CHK>"
"	<PARA1 Name='rPr_ECWScalMax' MIN='2.0' MAX='20.0' />"
"	<PARA2 Name='rPr_EngLubOilScalMax' MIN='5.0' MAX='20.0' />"
"	<PARA3 Name='rU_Gen_Nom[1]' MIN='70' MAX='65000' />"
"	<PARA4 Name='rF_Nom[1]' MIN='48.0' MAX='62.0' />"
"	<PARA5 />"
"</PARAMETER_CHK>"
;
; Statement, that this modules parameter check passing is mandatory (HA is allways mandatory, so other statements than TRUE here in this module are not possible)
"<MANDATORYMODULE>TRUE</MANDATORYMODULE>"
;
; Permanent Datamodule Filenames<!-- enter filenames for counter and INTERNAL parameter only; filename without extention-->
"<DATAMODULES>" ;<!-- optional; mehrere DATAMODULES erlaubt-->
"	<DATAMODULE>par_HA</DATAMODULE>"
"</DATAMODULES>"
;
; Dependencies Modules (MMxx.yy.zz.cc)
"<DEPENDENCIES>"
"	<DEPENDENCY MODULE='AB' VERSION='04.00.00.00' />"
"	<DEPENDENCY MODULE='AG' VERSION='04.14.00.00' />"
"	<DEPENDENCY MODULE='CU' VERSION='04.14.00.00' />"
"	<DEPENDENCY MODULE='EC' VERSION='04.14.00.00' />"
"	<DEPENDENCY MODULE='EX' VERSION='04.05.00.00' />"
"	<DEPENDENCY MODULE='GC' VERSION='04.14.00.00' />"
"	<DEPENDENCY MODULE='GD' VERSION='04.05.00.00' />"
"	<DEPENDENCY MODULE='GM' VERSION='04.01.00.00' />"
"	<DEPENDENCY MODULE='GR' VERSION='04.13.00.00' />"
"	<DEPENDENCY MODULE='GT' VERSION='04.10.00.00' />"
"	<DEPENDENCY MODULE='HC' VERSION='04.14.00.00' />"
"	<DEPENDENCY MODULE='IC' VERSION='04.05.00.00' />"
"	<DEPENDENCY MODULE='IG' VERSION='04.00.00.00' />"
"	<DEPENDENCY MODULE='KL' VERSION='04.05.00.00' />"
"	<DEPENDENCY MODULE='KN' VERSION='04.01.00.00' />"
"	<DEPENDENCY MODULE='MO' VERSION='04.05.00.00' />"
"	<DEPENDENCY MODULE='OP' VERSION='04.04.00.00' />"
"	<DEPENDENCY MODULE='PB' VERSION='04.03.00.00' />"
"	<DEPENDENCY MODULE='SA' VERSION='04.05.00.00' />"
"	<DEPENDENCY MODULE='SY' VERSION='04.13.00.00' />"
"	<DEPENDENCY MODULE='TR' VERSION='04.14.00.00' />"
"	<DEPENDENCY MODULE='VE' VERSION='04.04.00.00' />"
"	<DEPENDENCY MODULE='EM' VERSION='04.06.00.00' />"
"	<DEPENDENCY MODULE='EG' VERSION='04.25.00.00' />"    ; corrected for SW download via HMI
"   <DEPENDENCY VISVERSION='02.15.00.00' />"			; Dependencies Visualization
"</DEPENDENCIES>"
;
; Module function description
"<MODULEFUNCTION>" ;<!-- short overview documentation of module function; add reference to detailed information, if available-->
"	<General>	"
"	Engine Controller "
"	</General>	"
""
"	<F1 Name='Read & write IOs' LastModified='04.00.0.0'>"
"	controller for throttle and compressor bypass valve	"
"	</F1>"
"	<F2 Name='Scaling of IOs' LastModified='04.00.0.0'>"
"	 Abstract physical value to the needed raw value of different IO suppliers.	"
"	</F2>"
"	<F3 Name='Filter analog signals' LastModified='04.00.0.0'>"
"	 Filter analog inputs before the were used in the different modules.	"
"	</F3>"
"	<F4 Name='Signal qualitiy check' LastModified='04.00.0.0'>"
"	Check analog input signals if they are in a configured range.	"
"	</F4>"
"	<F5 Name='Hardware monitoring' LastModified='04.00.0.0'>"
"	Check if the hardware configuration maches to the detected IO modules.	"
"	</F5>"
"	<F6 Name='Initiate CAN communication' LastModified='04.00.0.0'>"
"	Initiate CAN interface and start the CAN communication with each CAN device (SAFI, GMU, ...).	"
"	</F6>"
"	<F7 Name='Communication to Multi Measure Devices' LastModified='04.00.0.0'>"
"	Read out asynchron measure data and handle parameter transfer.	"
"	</F7>"
""
"	<Info>"
"   UPDATE V4.2.0	version + dependencies changed (IF change with array index 0 for compatibility with c-tasks)	"
"   UPDATE V4.07.0	MMD unbalanced load meter reset function	"
"		  31.07.2018	Schmid,	 trigger for unbalanced load meter reset added	"
"		  09.08.2018	Schmid,	 2nd low temperature charge cooling circuit added	"
"		  20.09.2018	Schmid,	 unused IOs deleted	"
"		  28.09.2018	Schmid,	 changed scaling for gearbox oil quality sensors "
"		  17.12.2018	Schmid,	 added hydraulic ECW pre-heating for type 3+4, separate iIdx_OMSS PVs for TC5 and TC7 "
"		  24.01.2018	Schmid,	 changes on unbalanced load meter reset "
"		  22.03.2019	Schmid,	 gearbox oil quality sensor removed "
"		  29.03.2019	Schmid,	 bugfix: MMD does NOT restart IF powerlink is unplugged+plugged "
"								 wait for ModuleOk to activate AsIOAccRead/AsIOAccWrite FUBs "
" 	UPDATE V4.07.1 29.03.2019	Hohensinner,	Added IO: Execute_BS, removed IOs: P_Limit<x>Son_Gh "
"	UPDATE V4.07.2 15.05.2019	Schmid,	   coding guidelines: changed Para.rTi_Filt_LSL_In (datatype REAL) to Para.tiFilt_LSL_In (datatype TIME)"
"	UPDATE V4.07.3 01.08.2019	Zengerer,  vvm for gastrain added, META commets moved to XML Info section "
"	UPDATE V4.12.0 17.10.2022	Zengerer,  L_FreshOilTank, L_WasteOilTank, L_DayOilTank added "
"	UPDATE V4.14.0 25.11.2024	Zengerer,  Multi analog temp input variants: T_HW_Re, T_HW_ReAfEC, T_HW_Su +4 new type variant para "
"	</Info>"
""
"	<Customized LastModified='04.00.0.1'>	"
"	- HalIO Module is allways customized according to individual IO setup "
"	</Customized>	"
""
"</MODULEFUNCTION>"
;
"</META>"
```

### Module_HA.typ - HalIO Package data types
```iecst
(********************************************************************
 * COPYRIGHT -- INNIO Company
 ********************************************************************
 * Package: HAL_IO
 * File: HAL_IO.typ
 * Author: 105046866
 * Created: August 23, 2011
 ********************************************************************
 * Data types of package HAL_IO
 ********************************************************************)

TYPE
	tVIS2MM : 	STRUCT
		rP_WorkAct : ARRAY[0..2]OF REAL; (* counter for last produced work  *) (* OldName:slWorkAct; Cycle: *)
		rQ_WorkReac : ARRAY[0..2]OF REAL; (* counter last reactive engine work *) (* OldName:slWorkReac; Cycle: *)
		rP_WorkActRet : ARRAY[0..2]OF REAL; (* counter for last received work  *) (* OldName:slWorkActRet; Cycle: *)
		rQ_WorkReacRet : ARRAY[0..2]OF REAL; (* counter last received reactive engine work  *) (* OldName:slWorkReacRet; Cycle: *)
		bMMD2_Reset_Vis : BOOL; (* Reset of saved max values of MMDsynch 2 from visualization *) (* OldName:bResetMMU2Vis; Cycle: *)
		iEngID : DINT; (*Para: engine ID number*) (*OldName:new PV; Cycle: *)
		bCANCntReset : BOOL; (* CAN error counter value reset *)
		bMMD_UnbLoadReset : BOOL; (*Unbalanced load meter counter reset*) (*OldName:new PV; Cycle:*)
		tPlantComm : tPlantComm_VIS2MM; (*Datapoints for the Plant Communication*)
	END_STRUCT;
	tMM2VIS : 	STRUCT
		rI_MaxL1 : ARRAY[0..2]OF REAL; (* max. generator current phase 1 [A]  *) (* OldName:ssIMaxL1; Cycle: *)
		rI_MaxL2 : ARRAY[0..2]OF REAL; (* max. generator current phase 2 [A]  *) (* OldName:ssIMaxL2; Cycle: *)
		rI_MaxL3 : ARRAY[0..2]OF REAL; (* max. generator current phase 3 [A]  *) (* OldName:ssIMaxL3; Cycle: *)
		rP_ActMax : ARRAY[0..2]OF REAL; (* max. electric power [kW] *) (* OldName:ssPActMax; Cycle: *)
		rI_NMax : ARRAY[0..2]OF REAL; (* max. neutral current [A]  *) (* OldName:ssINMax; Cycle: *)
		rI_GenUnbalanced : ARRAY[0..2]OF REAL; (* unbalanced generator current [1/10 %]  *) (* OldName:ssIGenUnbalanced; Cycle: *)
		rF_MMD : ARRAY[0..2]OF REAL; (* frequency multi measure device *) (* OldName:ssFreq; Cycle: *)
		rF_MMD_Diff : ARRAY[0..2]OF REAL; (* frequency differenz system 1 / 2 *) (* OldName:ssFreqDiff; Cycle: *)
		rF_MMD_Synch1 : ARRAY[0..2]OF REAL; (* frequency sync-system 1  *) (* OldName:usSynch1Frequency; Cycle: *)
		rF_MMD_Synch2 : ARRAY[0..2]OF REAL; (* frequency sync-system 2 *) (* OldName:usSynch2Frequency; Cycle: *)
		rF_MMD_BusBar : ARRAY[0..2]OF REAL; (* frequency bus bar *) (* OldName:newPv; Cycle: *)
		rI_L1 : ARRAY[0..2]OF REAL; (* current 1 *) (* OldName:ssIL1; Cycle: *)
		rI_L2 : ARRAY[0..2]OF REAL; (* current 2 *) (* OldName:ssIL2; Cycle: *)
		rI_L3 : ARRAY[0..2]OF REAL; (* current 3 *) (* OldName:ssIL3; Cycle: *)
		rI_Avg : ARRAY[0..2]OF REAL; (* current average *) (* OldName:ssIAvg; Cycle: *)
		rI_Dyn : ARRAY[0..2]OF REAL; (* current dynamic *) (* OldName:usIDyn; Cycle: *)
		rI_N : ARRAY[0..2]OF REAL; (* current neutral *) (* OldName:ssIN; Cycle: *)
		rP_Act : ARRAY[0..2]OF REAL; (* power active */all *) (* OldName:ssPAct; Cycle: *)
		rP_ActUnfilt : ARRAY[0..2]OF REAL; (* power active */all *) (* OldName:ssPAct; Cycle: *)
		rS_Act : ARRAY[0..2]OF REAL; (* power apperent *) (* OldName:ssPApper; Cycle: *)
		rQ_Act : ARRAY[0..2]OF REAL; (* power reactive *) (* OldName:ssPReac; Cycle: *)
		rPF_Act : ARRAY[0..2]OF REAL; (* power factor *) (* OldName:ssCosPhi; Cycle: *)
		rU_L1N : ARRAY[0..2]OF REAL; (* voltage 1 *) (* OldName:ssUL1N; Cycle: *)
		rU_L1L2 : ARRAY[0..2]OF REAL; (* voltage 12 *) (* OldName:ssUL1L2; Cycle: *)
		rU_L2N : ARRAY[0..2]OF REAL; (* voltage 2 *) (* OldName:ssUL2N; Cycle: *)
		rU_L2L3 : ARRAY[0..2]OF REAL; (* voltage 23 *) (* OldName:ssUL2L3; Cycle: *)
		rU_L3N : ARRAY[0..2]OF REAL; (* voltage 3 *) (* OldName:ssUL3N; Cycle: *)
		rU_L3L1 : ARRAY[0..2]OF REAL; (* voltage 31 *) (* OldName:ssUL3L1; Cycle: *)
		rU_Avg : ARRAY[0..2]OF REAL; (* voltage average *) (* OldName:ssUAvg; Cycle: *)
		rAng_MMD_Diff : ARRAY[0..2]OF REAL; (* angle deviation synchronization *) (* OldName:ssSynchAngleDeviation; Cycle: *)
		iIdx_MMD_SynchMode : ARRAY[0..2]OF INT; (* synchronization mode *) (* OldName:usVisSynchMode; Cycle: *)
		rMMD_HW_Version : ARRAY[0..2]OF REAL; (* program version MMD *) (* OldName:usMMUSynchHWVariant; Cycle: *)
		rMMD_FW_Version : ARRAY[0..2]OF REAL; (* program version MMD firmware *) (* OldName:usMMUSynchFWVers; Cycle: *)
		rU_MMD_Diff : ARRAY[0..2]OF REAL; (* votage deviation synchronization *) (* OldName:ssSynchVoltDeviation; Cycle: *)
		rU_MMD_Synch1 : ARRAY[0..2]OF REAL; (* synchronization voltage 1 *) (* OldName:ssSynch1Volt; Cycle: *)
		rU_MMD_Synch2 : ARRAY[0..2]OF REAL; (* synchronization voltage 2 *) (* OldName:ssSynch2Volt; Cycle: *)
		rU_Bus_L1_2 : ARRAY[0..2]OF REAL; (* bus bar voltage 1 2 *) (* OldName:ssBusVoltPh1_2; Cycle: *)
		rU_Bus_L2_3 : ARRAY[0..2]OF REAL; (* bus bar voltage 2 3 *) (* OldName:ssBusVoltPh2_3; Cycle: *)
		rU_Bus_L3_1 : ARRAY[0..2]OF REAL; (* bus bar voltage 3 1 *) (* OldName:ssBusVoltPh3_1; Cycle: *)
		rU_Bus_L1N : ARRAY[0..2]OF REAL; (* bus bar voltage 1 *) (* OldName:ssBusVoltPh1_N; Cycle: *)
		rU_Bus_L2N : ARRAY[0..2]OF REAL; (* bus bar voltage 2 *) (* OldName:ssBusVoltPh2_N; Cycle: *)
		rU_Bus_L3N : ARRAY[0..2]OF REAL; (* bus bar voltage 3 *) (* OldName:ssBusVoltPh3_N; Cycle: *)
		bMMD_SynchDO : ARRAY[0..2]OF BOOL; (* feedback synch DO *) (* OldName:new PV; Cycle: *)
		bMsg3311 : BOOL; (* IO Channel Failure *) (* OldName:bAllModulesOK; Cycle: *)
		bMsg2399 : BOOL; (* A2399 - Shut down test bench priority 2 *)
		bMsg2400 : BOOL; (* A2400 - Shut down test bench priority 3 *)
		bMsg9400 : BOOL; (* W9400 - Warning test bench *)
		bMsg9384 : BOOL; (*Plant Communication Configuration failed*)
		bMsg9386 : BOOL; (*Plant Communication Interrupted*)
		bMsg9391 : BOOL; (*Plant Communication force active*)
		rUDiffMaxScale : ARRAY[0..2]OF REAL; (* Max scale value for voltage difference for synchronization *) (* OldName:new PV; Cycle: *)
		rF_DiffMaxScale : ARRAY[0..2]OF REAL; (* Max scale value for  frequence difference for synchronization *) (* OldName:new PV; Cycle: *)
		rF_DiffMinScale : ARRAY[0..2]OF REAL; (* Min scale value for  frequence difference for synchronization *) (* OldName:new PV; Cycle: *)
		bMO_SaftyLoop : BOOL; (* MORIS Safety loop signal *) (* OldName:new PV; Cycle: *)
		iCAN_HW_Slot : INT; (* CAN Module Socket Position Index *)
		sCAN_HW_WG : STRING[50]; (* Slot CAN Module - Wastegate actuators*)
		sCAN_HW_NOxS_IF1 : STRING[50]; (* Slot CAN Module - NOx sensor interface 1*)
		sCAN_HW_NOxS_IF2 : STRING[50]; (* Slot CAN Module - NOx sensor interface 2*)
		sCAN_HW_NOxS_IF3 : STRING[50]; (* Slot CAN Module - NOx sensor interface 3*)
		sCAN_HW_Slot_IPC : STRING[50]; (* Slot CAN Module - IPC PPC900 *)
		sCAN_HW_Slot_IPC_CMaU : STRING[50]; (* Slot CAN Module - IPC CM&U *)
		sCAN_HW_Slot_IPC_GE_IP : STRING[50]; (* Slot CAN Module - IPC GE-IP *)
		sCAN_HW_Slot_IPC_J920 : STRING[50]; (* Slot CAN Module - IPC J920 *)
		sCAN_HW_Slot_IPC_GE_IP_J920 : STRING[50]; (* Slot CAN Module - IPC GE-IP J920 *)
		sCAN_HW_Slot_IPC_3100 : STRING[50]; (* Slot CAN Module - IPC PPC3100 *)
		sCAN_HW_Slot_IPC_3100_J920 : STRING[50]; (* Slot CAN Module - IPC PPC3100 J920 *)
		sCAN_HW_Slot_X20CP368xX : STRING[50]; (* Slot CAN Module - X20CP368xX *)
		sCAN_HW_Slot_X20CP368xX_J920 : STRING[50]; (* Slot CAN Module - X20CP368xX J920 *)
		iCANopen_CMS_status : UINT; (* CAN Module Open CMS Status *)
		iCANopen_CMS_info : UINT; (* CAN Module Open CMS Info *)
		iCANopen_WG_status : UINT; (* CAN open status - Wastegate actuators*)
		iCANopen_NOxS_IF1_status : UINT; (* CAN open status - NOx sensor interface 1*)
		iCANopen_NOxS_IF2_status : UINT; (* CAN open status - NOx sensor interface 2*)
		iCANopen_NOxS_IF3_status : UINT; (* CAN open status - NOx sensor interface 3 *)
		iCMSmain_Init_status : UINT; (* CAN Module Main Init Status *)
		iSAFI_AllErrEventMax : UINT; (* SAFI All Modules Communication Error Event Max *)
		iSAFI_AllErrMaxCur : UINT; (* SAFI All Modules Communication Error Max Current *)
		iSAFI_AllErrMax : UINT; (* SAFI All Modules Communication Error Max All *)
		iSAFI_AllPhaseCntMax : UINT; (* SAFI All Modules Phase Counter Max *)
		iSAFI_AllErrAvgMax : UINT; (* SAFI All Modules Communication Error Average *)
		iSAFI_ErrEventMax : ARRAY[0..12]OF UINT; (* SAFI Communication Error Event Max *)
		iSAFI_ErrMaxCur : ARRAY[0..12]OF DINT; (* SAFI Communication Error Max Current *)
		iSAFI_ErrMax : ARRAY[0..12]OF UINT; (* SAFI Communication Error Max All *)
		iSAFI_PhaseCnt : ARRAY[0..12]OF UINT; (* SAFI Communication Phase Count *)
		iSAFI_ErrAvgCnt : ARRAY[0..12]OF UINT; (* SAFI Communication Error Average Count per Hour *)
		iTecJet_AllErrEventMax : UINT; (* TecJet All Modules Communication Error Event Max *)
		iTecJet_AllErrCount : UINT; (* TecJet All Modules Communication Error Count *)
		iTecJet_AllErrSlowMax : UINT; (* TecJet All Modules Communication Error Slow Max *)
		iTecJet_AllSlowPhaseCnt : UINT; (* TecJet All Modules Slow Phase Count *)
		iTecJet_AllErrSlowAvg : UINT; (* TecJet All Modules Communication Error Average *)
		iTecJet_ErrEventMax : ARRAY[0..4]OF UINT; (* TecJet Communication Error Event Max *)
		iTecJet_ErrMaxCur : ARRAY[0..4]OF UINT; (* TecJet Communication Error Max Current *)
		iTecJet_ErrMax : ARRAY[0..4]OF UINT; (* TecJet Communication Error Max All *)
		iTecJet_PhaseCnt : ARRAY[0..4]OF UINT; (* TecJet Communication Phase Count *)
		iTecJet_ErrAvgCnt : ARRAY[0..4]OF UINT; (* TecJet Communication Error Average Count per hour *)
		iKLS98_AllErrEventMax : UINT; (* KLS98 All Modules Communication Error Event Max *)
		iKLS98_AllErrMaxCur : UINT; (* KLS98 All Modules Communication Error Max Current *)
		iKLS98_AllErrMax : UINT; (* KLS98 All Modules Communication Error Max *)
		iKLS98_AllPhaseCntMax : UINT; (* KLS98 All Modules Phase Count Max *)
		iKLS98_AllErrAvgMax : UINT; (* KLS98 All Modules Communication Error Average Max *)
		iKLS98_ErrEventMax : ARRAY[0..24]OF UINT; (* KLS98 Communication Error Event Max *)
		iKLS98_ErrMaxCur : ARRAY[0..24]OF UINT; (* KLS98 Communication Error Max Current *)
		iKLS98_ErrMax : ARRAY[0..24]OF UINT; (* KLS98 Communication Error Max All *)
		iKLS98_PhaseCnt : ARRAY[0..24]OF UINT; (* KLS98 Communication Phase Count *)
		iKLS98_ErrAvgCnt : ARRAY[0..24]OF UINT; (* KLS98 Communication Error Average Count per hour *)
		iIC900_AllErrEventMax : UINT; (* IC900 All Modules Communication Error Event Max *)
		iIC900_AllErrCount : UINT; (* IC900 All Modules Communication Error Count *)
		iIC900_AllErrMax : UINT; (* IC900 All Modules Communication Error Max *)
		iIC900_AllPhaseCnt : UINT; (* IC900 All Modules Phase Count *)
		iIC900_AllErrAvg : UINT; (* IC900 All Modules Communication Error Average *)
		iMonic_AllErrEventMax : UINT; (* Monic All Modules Communication Error Event Max *)
		iMonic_AllErrCount : UINT; (* Monic All Modules Communication Error Max Current *)
		iMonic_AllErrMax : UINT; (* Monic All Modules Communication Error Max *)
		iMonic_AllPhaseCnt : UINT; (* Monic All Modules Phase Count *)
		iMonic_AllErrAvg : UINT; (* Monic All Modules Communication Error Average *)
		rUnbLoadMeter : ARRAY[0..2]OF REAL; (* unbalanced load meter [%] *) (* OldName:newPV; Cycle: *)
		sMMD_SerialNumber : ARRAY[0..2]OF STRING[11]; (* MMD Serial number *)
		iNum_CyleTimeViolCnt : UINT; (*Number of cylic time violations of TC#1*)
		tPlantComm : tPlantComm_MM2VIS; (*Datapoints for the Plant Communication*)
	END_STRUCT;
	ModulCfg_typ : 	STRUCT
		Used : BOOL;
		OK : BOOL;
		SlotNr : USINT;
		SubslotNr : USINT;
		StatusInfo : UINT;
		StatusWait : UINT;
		NodeNr : UINT;
		pModulOkPv : UDINT;
	END_STRUCT;
	ModulOK_typ : 	STRUCT
		ModuleOK : ARRAY[0..253]OF BOOL;
	END_STRUCT;
	StationCfg_typ : 	STRUCT
		Modul : ARRAY[0..49]OF ModulCfg_typ;
	END_STRUCT;
	CanDeviceGo : 	STRUCT
		CANDevGo : ARRAY[0..1]OF USINT;
		ECANDevGo : USINT;
	END_STRUCT;
	ModulID_Type : 	STRUCT
		iID : INT;
		iXX : INT;
		iYY : INT;
		iZZ : INT;
		iCC : INT;
	END_STRUCT;
	OUT_HA_struct : 	STRUCT
		tHA2AB : MM2AmmBase; (* HalIO module to AMM base data transfer *) (* OldName:new PV; Cycle:2 *)
		iECanDevGo : USINT; (* event status CAN device go *) (* OldName:new PV; Cycle:2 *)
		iCANIdent : UDINT; (* CAN open ident *) (* OldName:new PV; Cycle:2 *)
		iCANIdentIGN2 : UDINT; (* CAN open ident *) (* OldName:new PV; Cycle:2 *)
		tHA2PB : MM2ParaBase_type; (* Data exchange structure to ParaBase *) (* OldName:new PV; Cycle:5 *)
		iGM1_MStepActPos : DINT; (*gasmixer 1 - Actual position from SM1426-Module [Microsteps]*) (*OldName: slGM1_MStepActPos_TC1; Cycle: 5;*)
		iGM1_Status : UINT; (*gasmixer 1 - Status Word from SM1426-Module*) (*OldName: usGM1_Status_TC1; Cycle: 5;*)
		iGM2_MStepActPos : DINT; (*gasmixer 2 - Actual position from SM1426-Module [Microsteps]*) (*OldName: slGM2_MStepActPos_TC1; Cycle: 5;*)
		iGM2_Status : UINT; (*gasmixer 2 - Status Word from SM1426-Module*) (*OldName: usGM2_Status_TC1; Cycle: 5;*)
		tModulID : ModulID_Type; (* HalIO module ID *) (* OldName:new PV; Cycle:5 *)
		iCAN_CB_us_ident : UDINT; (*CAN user ident for conrod bearing system*) (* OldName:new PV; Cycle:8*)
		bSimWinMOD_Active : BOOL; (* WinMode simulation active *) (* OldName:new PV; Cycle:5*)
		szEng_Motorversion : STRING[17]; (* Para: Engine version *) (* OldName:new PV; Cycle:8*)
		szOrderID : STRING[17]; (*Para: application ID string*) (* OldName:szApplication; Cycle:8*)
		iEngID : DINT; (*Para: engine ID number*) (* OldName:new PV; Cycle:8*)
		iCAN_NOxS_IF1_us_ident : UDINT; (*User ident for NOx sensor CAN interface 1*) (* OldName:new PV; Cycle:8*)
		rI_MaxL1 : ARRAY[0..2]OF REAL; (* max. generator current phase 1 [A]  *) (* OldName:ssIMaxL1; Cycle: 5*)
		rI_MaxL2 : ARRAY[0..2]OF REAL; (* max. generator current phase 2 [A]  *) (* OldName:ssIMaxL2; Cycle: 5*)
		rI_MaxL3 : ARRAY[0..2]OF REAL; (* max. generator current phase 3 [A]  *) (* OldName:ssIMaxL3; Cycle: 5*)
		iCAN_NOxS_IF2_us_ident : UDINT; (*User ident for NOx sensor CAN interface 2*) (* OldName:new PV; Cycle:8*)
		iCAN_NOxS_IF3_us_ident : UDINT; (*User ident for NOx sensor CAN interface 3*) (* OldName:new PV; Cycle:8*)
		szPB1_DeviceName : STRING[40]; (*Device adress from I/O Module Profibus slave 1*) (* OldName:new PV; Cycle:8*)
		szPB2_DeviceName : STRING[40]; (*Device adress from I/O Module Profibus slave 1*) (* OldName:new PV; Cycle:8*)
		szPN_DeviceName : STRING[40]; (*Device adress from I/O Module Profinet*) (* OldName:new PV; Cycle:8*)
		szMBRTU_DeviceName : STRING[40]; (*Device adress from I/O Module Modbus RTU*) (* OldName:new PV; Cycle:8*)
		szMBTCP_DeviceName : STRING[40]; (*Device adress from I/O Module Modbus TCP*) (* OldName:new PV; Cycle:8*)
		bSimWinMOD_FastStart : BOOL; (* WinMode fast start of engine*) (* OldName:new PV; Cycle:5*)
		iSerialNumber_CPU : UDINT; (*Serial number CPU*) (*OldName:new PV; Cycle:5;*)
		iModulID_CPU : UINT; (*Modul ID CPU*) (*OldName:new PV; Cycle:5;*)
		iPowerOnCycles : UDINT; (*Power On cycles CPU*) (*OldName:new PV; Cycle:5;*)
		iOperatingHours_CPU : UDINT; (*Operating hours CPU*) (*OldName:new PV; Cycle:5;*)
		iBatterieStatus : USINT; (*Batterie Status IPC*) (*OldName:new PV; Cycle:5;*)
		iT_CPU : UINT; (*Temperature CPU*) (*OldName:new PV; Cycle:5;*)
		iT_CPU_PLC : UINT; (*Temperature X20CP368xX CPU*) (*OldName:new PV; Cycle:5;*)
		iT_Board : UINT; (*Temperature Board*) (*OldName:new PV; Cycle:5;*)
		iT_Chipset : UINT; (*Temperature Chipset*) (*OldName:new PV; Cycle:5;*)
		iT_PS : UINT; (*Temperature IPC board power supply*) (*OldName:new PV; Cycle:5;*)
		iT_CFast : UINT; (*Temperature IPC CFast*) (*OldName:new PV; Cycle:5;*)
		bSimWinMOD_withoutBus_Active : BOOL; (*WinMode simulation without Bus Hardware active *) (*OldName:new PV; Cycle:5*)
		bCANCntReset : BOOL; (* CAN error counter value reset *) (*OldName: bCANCounterReset; Cycle:5;*)
		rAng_MMD_Diff : ARRAY[0..2]OF REAL; (* angle deviation synchronization *) (* OldName:ssSynchAngleDeviation; Cycle: 1*)
		tHW_Switches : OpMode_Switches; (*Hardware operation mode switches*)
		rCustomizedHA : ARRAY[0..300]OF REAL; (*New customizable interface 2017  - BETA PHASE, use only in coordination with TPSS*)
		rI_Dyn : ARRAY[0..2]OF REAL; (* current dynamic *) (* OldName:usIDyn; Cycle: *)
		rI_GenUnbalanced : ARRAY[0..2]OF REAL; (* unbalanced generator current [1/10 %]  *) (* OldName:ssIGenUnbalanced; Cycle: *)
		rU_MMD_Diff : ARRAY[0..2]OF REAL; (* votage deviation synchronization *) (* OldName:ssSynchVoltDeviation; Cycle: *)
		iIdx_MMD_SynchMode : ARRAY[0..2]OF INT; (* synchronization mode *) (* OldName:usVisSynchMode; Cycle: *)
		iT_CFast2 : UINT; (*Temperature IPC CFast 2*) (*OldName:new PV; Cycle:5;*)
		iSystemTime : DINT; (*System time for exception task logic*)
		iCAN_OQS_OC_us_ident : UDINT; (*User ident for OQS OC sensor CAN interface*) (* OldName:new PV; Cycle:2*)
		iCAN_WG_us_ident : UDINT; (*User ident for WasteGate CAN interface*)
		szMBTCP1_DeviceName : STRING[40]; (*Device adress from I/O Module Modbus TCP*)
		szMBTCP2_DeviceName : STRING[40]; (*Device adress from I/O Module Modbus TCP Slave coupling 2*) (* OldName:new PV; Cycle:8*)
		szMBTCP3_DeviceName : STRING[40]; (*Device adress from I/O Module Modbus TCP Master *) (* OldName:new PV; Cycle:8*)
		bTOF_HwBypassDigitalTwin : BOOL; (*Hardware bypass digital twin - T3 adaptive cranking time*)
		tPlantCom_M2E_In_Cust100ms : ARRAY[0..4]OF tPlantComData_Cust100ms; (*PlantCom Customized Data M2E_In_100ms*)
		tPlantCom_E2E_In_Cust100ms : ARRAY[0..32]OF tPlantComData_Cust100ms; (*PlantCom Customized Data E2E_In_100ms*)
		tPlantCom_E2E_In_Cust10ms : ARRAY[0..32]OF tPlantComData_Cust10ms; (*PlantCom Customized Data E2E_In_10ms*)
		tPlantCom_M2E_In_Cust10ms : ARRAY[0..4]OF tPlantComData_Cust10ms; (*PlantCom Customized Data M2E_In_10ms*)
		bPlantComCfgOk : BOOL;
	END_STRUCT;
	IN_HA_struct : 	STRUCT
		bEng_Dem : BOOL; (* module demanded *) (* OldName:M_AGFD; Cycle:5 *)
		tAB2HA : AmmBase2MM; (* AMM base to SAFI data transfer *) (* OldName:QUITT_WA; Cycle:2 *)
		tEng_Run : HALioDo_Type; (* engine operating state *) (* OldName:M_BTRB; Cycle:5 *)
		bMMD2_Reset : BOOL; (* Reset of saved max values of MMDsynch 2 *) (* OldName:bResetMMU2; Cycle:5 *)
		bSyncSlipMode : ARRAY[0..2]OF BOOL; (* MMD synchronization with slip mode *) (* OldName:bSyncSlipMode; Cycle:5 *)
		tMonic_CanGo : CanDeviceGo; (* CAN device initializing *) (* OldName:new PV; Cycle:5 *)
		tSAFI_CanGo : CanDeviceGo; (* CAN device initializing *) (* OldName:new PV; Cycle:5 *)
		tICxx_CanGo : CanDeviceGo; (* CAN device initializing *) (* OldName:new PV; Cycle:5 *)
		tKLS98_CanGo : CanDeviceGo; (* CAN device initializing *) (* OldName:new PV; Cycle:5 *)
		tGasMeteringUnit_CanGo : CanDeviceGo; (* CAN device initializing *) (* OldName:new PV; Cycle:5 *)
		tPB2MM : ParaBase2MM_type; (* Data exchange structure to ParaBase *) (* OldName:new PV; Cycle:5 *)
		iGM1_Control : UINT; (*gasmixer 1 - Handover Control Word to SM1426-Module*) (*OldName: usGM1_Control_TC1; Cycle: 5;*)
		iGM1_Mode : SINT; (*gasmixer 1 - Handover Mode to SM1426-Module*) (*OldName: scGM1_Mode_TC1; Cycle: 5;*)
		iGM1_MStepSetPos : DINT; (*gasmixer 1 - Handover Set position to SM1426-Module [Microsteps]*) (*OldName: slGM1_MStepSetPos_TC1; Cycle: 5;*)
		iGM2_Control : UINT; (*gasmixer 2 - Handover Control Word to SM1426-Module*) (*OldName: usGM2_Control_TC1; Cycle: 5;*)
		iGM2_Mode : SINT; (*gasmixer 2 - Handover Mode to SM1426-Module*) (*OldName: scGM2_Mode_TC1; Cycle: 5;*)
		iGM2_MStepSetPos : DINT; (*gasmixer 2 - Handover Set position to SM1426-Module [Microsteps]*) (*OldName: slGM2_MStepSetPos_TC1; Cycle: 5;*)
		rN_EngAct : REAL; (*Engine Speed (1/min)*) (*OldName:ZDGSpeed; Cycle:5;*)
		bGCB_DemSy : BOOL; (*Demand synchronization generator circuit breaker *) (*OldName:ASYANW,gcb[1].dmnd_sy; Cycle:5;*)
		tILF_SOn : HALioDo_Type; (* DO: ILF switched on*)
		tILF_SOf : HALioDo_Type; (* DO: ILF switched off*)
		tFC_SOn : HALioDo_Type; (* DO: frequency control switched on*)
		tFC_SOf : HALioDo_Type; (* DO: frequency control switched off*)
		tPU_SOn : HALioDo_Type; (* DO: P(U) switched on*)
		tPU_SOf : HALioDo_Type; (* DO: P(U) switched off*)
		iCnt_OpHours : DINT; (* operating hours counter *) (*OldName:betrieb_h;Cycle:2;*)
		iIC900CommErrCount : USINT; (* comm. error counter *)
		iMonicCommErrCount : USINT; (* counter Communication error monic *)
		iTecJetCommErrCount : USINT; (* CAN TecJet All Modules Communication Error Count *)
		iE_IgnStat : USINT; (* events igniton system status *)
		iEMonStatus : USINT; (* event monic status *)
		tE_TEC : ARRAY[0..4]OF _tEventTEC; (* CAN events gas inject valve param. *)
		iTecErrCntMax : ARRAY[0..4]OF USINT; (* CAN TecJet Modules Communication max value for wrong gas flow trans *)
		iTecErrCnt : ARRAY[0..4]OF USINT; (* CAN TecJet Modules Communication counter for wrong gas flow transm. *)
		tE_KLS : ARRAY[0..24]OF _tEventKLS; (* CAN events KLS98 *)
		tE_SAFI : ARRAY[0..12]OF _tEventSAFI; (* SAFI CAN Events *)
		iCnt_SA_ComErr : ARRAY[0..12]OF DINT; (* SAFI communication error counter *) (* OldName:usSAFIComErrCnt; Cycle:  *)
		iKLS98CommErrCount : ARRAY[0..24]OF USINT; (* CAN KLS98 All Module Communication Error Count*)
		rCustomizedHA : ARRAY[0..300]OF REAL; (*New customizable interface 2017  - BETA PHASE, use only in coordination with TPSS*)
		iIdx_OMSS : INT; (*Index of operation mode selector switch 0  OFF, 1  MANUAL, 2  AUTOMATIC, 3 Test (Optional)*) (*OldName:BWS_HA,PROBE; Cycle:5;*)
		iIdx_OMSS_TC7 : INT; (*Index of operation mode selector switch 0  OFF, 1  MANUAL, 2  AUTOMATIC, 3 Test (Optional)*) (*OldName:BWS_HA,PROBE; Cycle:7;*)
		bMMD_GenAlarmTestOn : BOOL; (* MMD_Gen alarm test On *) (*OldName:newPv; Cycle:5;*)
		iSt_OpMode : UDINT; (*engine operation status*) (*OldName:newPv; Cycle:2;*)
		bFSync_NarrowSyncWin : BOOL; (* use narrow sync window if fast-sync controller is active *) (*OldName:newPv; Cycle:5;*)
		iModule : USINT; (*Engine Module Number*)
		iIdx_RSS : INT; (*Request Selector Switch*)
		iIdx_SyOMSS : INT; (*Synchronization Selector Switch*)
		rP_Nom : REAL; (*nominal electric power [KW], depends on gastype *)
		tPlantCom_E2E_Out_Cust100ms : tPlantComData_Cust100ms; (*PlantCom Customized Data E2E_Out_100ms*)
		tPlantCom_E2M_Out_Cust100ms : ARRAY[0..4]OF tPlantComData_Cust100ms; (*PlantCom Customized Data E2M_Out_100ms*)
		tPlantCom_E2E_Out_Cust10ms : tPlantComData_Cust10ms; (*PlantCom Customized Data E2E_Out_10ms*)
		tPlantCom_E2M_Out_Cust10ms : ARRAY[0..4]OF tPlantComData_Cust10ms; (*PlantCom Customized Data E2M_Out_10ms*)
		bSafetyPLC_Active : BOOL; (*SAFETY PLC: SafetyPLC is active*) (*OldName: new PV; Cycle: 5;*) (*V04.25.00.00*)
		bSafeOUT_SafetyLoop_EmStop : BOOL; (*SAFETY PLC: Safety loop - Emergency stop push button OK*) (*OldName: new PV; Cycle: 5;*) (*V04.25.00.00*)
		bSafeOUT_SafetyLoop_Eng : BOOL; (*SAFETY PLC: Safety loop - Engine OK*) (*OldName: new PV; Cycle: 5;*) (*V04.25.00.00*)
	END_STRUCT;
	_tEventTEC : 	STRUCT
		Conf : ARRAY[0..8]OF USINT;
		Data : ARRAY[0..5]OF USINT;
		Contr : ARRAY[0..1]OF USINT;
		Status : ARRAY[0..5]OF USINT;
	END_STRUCT;
	_tEventKLS : 	STRUCT
		conf : ARRAY[0..99]OF USINT;
	END_STRUCT;
	_tEventSAFI : 	STRUCT
		conf : ARRAY[0..35]OF USINT;
		zuend : ARRAY[0..1]OF USINT;
		error : USINT;
		sdata : ARRAY[0..4]OF USINT;
		idata : ARRAY[0..30]OF USINT;
		kdata : ARRAY[0..30]OF USINT;
		ddata : ARRAY[0..53]OF USINT;
		dmdata1 : ARRAY[0..5]OF USINT;
		kmdata : ARRAY[0..7]OF USINT;
		dmdata2 : ARRAY[0..15]OF USINT;
		smdata : ARRAY[0..9]OF USINT;
		status : ARRAY[0..11]OF USINT;
		bez : USINT;
		ref : USINT;
		cur : USINT;
		diag : ARRAY[0..18]OF USINT;
	END_STRUCT;
	OpMode_Switches : 	STRUCT
		iIdx_OMS_Hw : INT; (* index of hardware operation mode selector switch *)
		iIdx_RMS_Hw : INT; (* index of hardware request mode selector switch *)
		iIdx_SyOMS_Hw : INT; (* index of hardware synchronisation operation mode selector switch *)
		bGoodQual : BOOL; (* Global GoodQual Bit for all 3 hw-switches *)
	END_STRUCT;
	HALIO2CUSTOM_Struct : 	STRUCT
		tSet_LFSMO_DB_COn : HALioDi_Type; (*DI: Activation of LFSMO Deadband via AI*)
		tSet_LFSMO_DB_COf : HALioDi_Type; (*DI: De-activation of LFSMO Deadband via AI*)
		tSet_LFSMU_DB_COn : HALioDi_Type; (*DI: Activation of LFSMU Deadband via AI*)
		tSet_LFSMU_DB_COf : HALioDi_Type; (*DI: De-activation of LFSMU Deadband via AI*)
		tSet_LFSMO_Droop_COn : HALioDi_Type; (*DI: Activation of LFSMO Droop via AI*)
		tSet_LFSMO_Droop_COf : HALioDi_Type; (*DI: De-activation of LFSMO Droop via AI*)
		tSet_LFSMU_Droop_COn : HALioDi_Type; (*DI: Activation of LFSMO Droop via AI*)
		tSet_LFSMU_Droop_COf : HALioDi_Type; (*DI: De-activation of LFSMO Droop via AI*)
		tSet_FSMU_Droop_COn : HALioDi_Type; (*DI: Activation of FSMU Droop via AI*)
		tSet_FSMU_Droop_COf : HALioDi_Type; (*DI: De-activation of FSMU Droop via AI*)
		tSet_FSMO_Droop_COn : HALioDi_Type; (*DI: Activation of FSMO Droop via AI*)
		tSet_FSMO_Droop_COf : HALioDi_Type; (*DI: De-activation of FSMO Droop via AI*)
		tSet_FSMU_DB_COn : HALioDi_Type; (*DI: Activation of FSMU Deadband via AI*)
		tSet_FSMU_DB_COf : HALioDi_Type; (*DI: De-activation of FSMO Deadband via AI*)
		tSet_FSMO_DB_COn : HALioDi_Type; (*DI: Activation of FSMO Deadband via AI*)
		tSet_FSMO_DB_COf : HALioDi_Type; (*DI: De-activation of FSMO Deadband via AI*)
		tSet_FSM_RMC_Up_COn : HALioDi_Type; (*DI: Activation of positive Margin FSM via AI*)
		tSet_FSM_RMC_Up_COf : HALioDi_Type; (*DI: De-activation of positive Margin FSM via AI*)
		tSet_FSM_RMC_Down_COn : HALioDi_Type; (*DI: Activation of negative Margin FSM via AI*)
		tSet_FSM_RMC_Down_COf : HALioDi_Type; (*DI: De-activation of negative Margin FSM via AI*)
		tSet_U_Droop_COn : HALioDi_Type; (*DI: Activation of droop U via AI*)
		tSet_U_Droop_COf : HALioDi_Type; (*DI: De-activation of droop U via AI*)
		tSet_FSM_Rmp_COn : HALioDi_Type; (*DI: Activation of Ramp rate via AI*)
		tSet_FSM_Rmp_COf : HALioDi_Type; (*DI: De-activation of Ramp rate via AI*)
		tSet_F_Ref_FSM_COn : HALioDi_Type; (*DI: Activation of Reference frequency for FSM/LFSM via AI*)
		tSet_F_Ref_FSM_COf : HALioDi_Type; (*DI:De-activation of Reference frequency for FSM/LFSM via AI*)
		bCheck_HA2CU : BOOL; (* Controlbit for HALio to Custom structure *)
	END_STRUCT;
	HALIO2GRID_Struct : 	STRUCT
		tF_LFSMO_DB : HALioAi_Type; (* LFSMO Deadband from EU [Hz] *)
		tF_LFSMU_DB : HALioAi_Type; (* LFSMU Deadband from EU [Hz] *)
		tF_LFSMO_Droop : HALioAi_Type; (* LFSMO Droop from EU [Hz] *)
		tF_LFSMU_Droop : HALioAi_Type; (* LFSMU Droop from EU [Hz] *)
		tF_FSMU_Droop : HALioAi_Type; (* FSMU Droop from EU [Hz] *)
		tF_FSMO_Droop : HALioAi_Type; (* FSMO Droop from EU [Hz] *)
		tF_FSMU_DB : HALioAi_Type; (* FSMU Deadband from EU [Hz] *)
		tF_FSMO_DB : HALioAi_Type; (* FSMO Deadband from EU [Hz] *)
		tP_FSM_RMC_Up : HALioAi_Type; (* Positive Margin FSM from EU [%Pnom] *)
		tP_FSM_RMC_Down : HALioAi_Type; (* Negative Margin FSM from EU [%Pnom] *)
		tU_Droop : HALioAi_Type; (* U droop from EU [%] *)
		tFSM_Rmp_Up : HALioAi_Type; (* Ramp rate UP from EU [%Pnom/s] *)
		tFSM_Rmp_Down : HALioAi_Type; (* Ramp rate DOWN from EU [%Pnom/s] *)
		tF_Ref_FSM : HALioAi_Type; (* Reference frequency for FSM/LFSM from EU [Hz] *)
		tJunctionBox_GnlAlm : HALioDi_Type; (* DI:General Alarm from junction box *)
		bCheck_HA2GR : BOOL; (* Controlbit for HALio to Grid structure *)
	END_STRUCT;
	tPlantComm_MM2VIS : 	STRUCT
		iIO_Typ_Dir_Num_Min : USINT; (*First Asset of the Communication (Selection lower bound)*)
		iIO_Typ_Dir_Num_Max : USINT; (*Last Asset of the Communication (Selection upper bound)*)
		iFrc_Gbl : USINT; (*Numer of forced Signals from/to all assets*)
		iFrc_Act : USINT; (*Numer of forced Signals from/to the selected asset*)
		rInt : ARRAY[0..15]OF REAL; (*Intern Value (Processed by PLC) of the signal*)
		rExt : ARRAY[0..15]OF REAL; (*Extern Value (Transfered via OpcUA) of the signal*)
		iNum : ARRAY[0..15]OF USINT; (*Signal Number (Index)*)
		iComment : ARRAY[0..15]OF UINT; (*Signal Description e.g. Watchdog => Textenum*)
		bMas_Ena : ARRAY[0..4]OF BOOL; (*Bus Diagnostic: Master communication available*)
		bEng_Ena : ARRAY[0..32]OF BOOL; (*Bus Diagnostic: Engine communication available*)
		bCfg_OK : BOOL; (*OpcUA Confiugration OK*)
		bCfg_Err : BOOL; (*OpcUA Configuration Error*)
		bCfg_Rst : BOOL; (*OpcUA Configuration Change: Reboot Required*)
	END_STRUCT;
	tPlantComm_VIS2MM : 	STRUCT
		iIO_Typ : USINT; (*Selected IO Type: (AI, DI, AO, DO)*)
		iIO_Typ_Dir : USINT; (*Selected Signal Direction: From/To Master/Engine*)
		iIO_Typ_Dir_Num : USINT; (*Selected Asset e.g. Engine 3*)
		iNum_Start : USINT; (*First Signal to be displayed in the diagnostics table (Offset)*)
		bFrc_Gbl : BOOL; (*Unforce all Signals from/to all the assets*)
		bFrc_Act : BOOL; (*Unforce all Signals from/to the selected asset*)
		bFrc : ARRAY[0..15]OF BOOL; (*Force Active/Inactive of the displayed signals*)
		bFrc_Int : ARRAY[0..15]OF BOOL; (*Force Value for digital Signals*)
		rFrc_Int : ARRAY[0..15]OF REAL; (*Force Value for analog Signals*)
	END_STRUCT;
	tPlantComm_Para : 	STRUCT
		iMas_Num_Min : USINT; (*[Para 15022] First Master in the Communication*)
		iMas_Num_Max : USINT; (*[Para 15023] Last Master in the Communication*)
		iEng_Num_Min : USINT; (*[Para 15024] First Engine in the Communication*)
		iEng_Num_Max : USINT; (*[Para 15025] Last Engine in the Communication*)
		bActive : BOOL; (*[Para 15021] Plant Communication active*)
	END_STRUCT;
	tPlantComData_Cust10ms : 	STRUCT
		digitalSignals : ARRAY[0..15]OF tDigitalSignal_Struct;
		analogSignals : ARRAY[0..7]OF tAnalogSignal_Struct;
	END_STRUCT;
	tPlantComData_Cust100ms : 	STRUCT
		digitalSignals : ARRAY[0..31]OF tDigitalSignal_Struct;
		analogSignals : ARRAY[0..15]OF tAnalogSignal_Struct;
	END_STRUCT;
	tDigitalSignal_Struct : 	STRUCT
		Value : BOOL;
		GoodQual : BOOL;
	END_STRUCT;
	tAnalogSignal_Struct : 	STRUCT
		Value : REAL;
		GoodQual : BOOL;
	END_STRUCT;
END_TYPE
```
